(* IEC 61131-3 sources: SmartHomeNew/ (part 7) *)

(* ---- FB_Heating_Source_Stability_Observer.st ---- *)
// ==============================================================================
// Heating source stability observer
//
// Predictive observability-only layer.
//
// DOES NOT own runtime authority.
// DOES NOT own outputs.
// DOES NOT close valves.
// DOES NOT modify heating demand.
// DOES NOT override runtime decisions.
//
// Observes:
// - source switching frequency
// - fallback oscillation
// - degradation persistence
// - recovery trends
// - confidence volatility
//
// Publishes predictive instability semantics only.
//
// Reads only canonical runtime projection contracts.
// Does not depend on explainability publication topology.
// ==============================================================================
FUNCTION_BLOCK FB_Heating_Source_Stability_Observer
VAR_INPUT
    VI_Enable : BOOL;
    VI_System_Time_MS : UDINT;
END_VAR

VAR
    L_i : INT;

    L_Last_Confidence : ARRAY[1..GVL_CONSTANTS.C_MAX_HEATING_CIRCUITS] OF REAL;

    L_Confidence_Delta : REAL;
    L_Confidence_Volatility : REAL;
    L_Source_Trust_Trend : REAL;
    L_Instability_Score : REAL;
END_VAR

IF NOT VI_Enable THEN
    RETURN;
END_IF;

FOR L_i := 1 TO GVL_CONSTANTS.C_MAX_HEATING_CIRCUITS DO

    // ======================================================
    // VISIBILITY
    // ======================================================
    GVL_Heating_Source_Stability.G_State[L_i].Visible :=
        GVL_Heating_Runtime_Projection.G_Circuit_Projection[L_i].Visible;

    // ======================================================
    // EDGE COUNTING
    // ======================================================
    IF GVL_Heating_Runtime_Projection.G_Circuit_Projection[L_i].Source_Switched_Event THEN
        IF GVL_Heating_Source_Stability.G_State[L_i].Source_Switch_Count < 65535 THEN
            GVL_Heating_Source_Stability.G_State[L_i].Source_Switch_Count :=
                GVL_Heating_Source_Stability.G_State[L_i].Source_Switch_Count + 1;
        END_IF;

        GVL_Heating_Source_Stability.G_State[L_i].Last_Observation_MS :=
            VI_System_Time_MS;
    END_IF;

    IF GVL_Heating_Runtime_Projection.G_Circuit_Projection[L_i].Fallback_Activated_Event THEN
        IF GVL_Heating_Source_Stability.G_State[L_i].Fallback_Activation_Count < 65535 THEN
            GVL_Heating_Source_Stability.G_State[L_i].Fallback_Activation_Count :=
                GVL_Heating_Source_Stability.G_State[L_i].Fallback_Activation_Count + 1;
        END_IF;

        GVL_Heating_Source_Stability.G_State[L_i].Last_Observation_MS :=
            VI_System_Time_MS;
    END_IF;

    IF GVL_Heating_Runtime_Projection.G_Circuit_Projection[L_i].Fallback_Recovered_Event THEN
        IF GVL_Heating_Source_Stability.G_State[L_i].Fallback_Recovery_Count < 65535 THEN
            GVL_Heating_Source_Stability.G_State[L_i].Fallback_Recovery_Count :=
                GVL_Heating_Source_Stability.G_State[L_i].Fallback_Recovery_Count + 1;
        END_IF;

        GVL_Heating_Source_Stability.G_State[L_i].Last_Observation_MS :=
            VI_System_Time_MS;
    END_IF;

    IF GVL_Heating_Runtime_Projection.G_Circuit_Projection[L_i].Source_Loss_Event THEN
        IF GVL_Heating_Source_Stability.G_State[L_i].Source_Loss_Count < 65535 THEN
            GVL_Heating_Source_Stability.G_State[L_i].Source_Loss_Count :=
                GVL_Heating_Source_Stability.G_State[L_i].Source_Loss_Count + 1;
        END_IF;

        GVL_Heating_Source_Stability.G_State[L_i].Last_Observation_MS :=
            VI_System_Time_MS;
    END_IF;

    // ======================================================
    // CONFIDENCE VOLATILITY
    // ======================================================
    L_Confidence_Delta := ABS(
        GVL_Heating_Runtime_Projection.G_Circuit_Projection[L_i].Selected_Source_Confidence -
        L_Last_Confidence[L_i]
    );

    L_Confidence_Volatility :=
        GVL_Heating_Source_Stability.G_State[L_i].Confidence_Volatility * REAL#0.90 +
        L_Confidence_Delta * REAL#0.10;

    IF L_Confidence_Volatility < REAL#0.0 THEN
        L_Confidence_Volatility := REAL#0.0;
    ELSIF L_Confidence_Volatility > REAL#1.0 THEN
        L_Confidence_Volatility := REAL#1.0;
    END_IF;

    GVL_Heating_Source_Stability.G_State[L_i].Confidence_Volatility :=
        L_Confidence_Volatility;

    // ======================================================
    // SOURCE TRUST TREND
    // ======================================================
    L_Source_Trust_Trend :=
        GVL_Heating_Source_Stability.G_State[L_i].Source_Trust_Trend * REAL#0.95 +
        GVL_Heating_Runtime_Projection.G_Circuit_Projection[L_i].Selected_Source_Confidence * REAL#0.05;

    IF GVL_Heating_Runtime_Projection.G_Circuit_Projection[L_i].Source_Degraded THEN
        L_Source_Trust_Trend := L_Source_Trust_Trend * REAL#0.98;
    END_IF;

    IF L_Source_Trust_Trend < REAL#0.0 THEN
        L_Source_Trust_Trend := REAL#0.0;
    ELSIF L_Source_Trust_Trend > REAL#1.0 THEN
        L_Source_Trust_Trend := REAL#1.0;
    END_IF;

    GVL_Heating_Source_Stability.G_State[L_i].Source_Trust_Trend :=
        L_Source_Trust_Trend;

    // ======================================================
    // TREND OBSERVATION
    // ======================================================
    GVL_Heating_Source_Stability.G_State[L_i].Degraded_Trend_Visible :=
        GVL_Heating_Runtime_Projection.G_Circuit_Projection[L_i].Source_Degraded OR
        (GVL_Heating_Source_Stability.G_State[L_i].Fallback_Activation_Count >
         GVL_Heating_Source_Stability.G_State[L_i].Fallback_Recovery_Count);

    GVL_Heating_Source_Stability.G_State[L_i].Recovery_Trend_Visible :=
        (GVL_Heating_Source_Stability.G_State[L_i].Fallback_Recovery_Count > 0) AND
        (GVL_Heating_Source_Stability.G_State[L_i].Fallback_Recovery_Count >=
         GVL_Heating_Source_Stability.G_State[L_i].Fallback_Activation_Count);

    GVL_Heating_Source_Stability.G_State[L_i].Oscillation_Detected :=
        (GVL_Heating_Source_Stability.G_State[L_i].Source_Switch_Count >= 3) OR
        ((GVL_Heating_Source_Stability.G_State[L_i].Fallback_Activation_Count >= 2) AND
         (GVL_Heating_Source_Stability.G_State[L_i].Fallback_Recovery_Count >= 2));

    // ======================================================
    // INSTABILITY SCORE
    // ======================================================
    L_Instability_Score := REAL#0.0;

    IF GVL_Heating_Source_Stability.G_State[L_i].Oscillation_Detected THEN
        L_Instability_Score := L_Instability_Score + REAL#40.0;
    END_IF;

    IF GVL_Heating_Source_Stability.G_State[L_i].Degraded_Trend_Visible THEN
        L_Instability_Score := L_Instability_Score + REAL#30.0;
    END_IF;

    IF GVL_Heating_Source_Stability.G_State[L_i].Source_Loss_Count > 0 THEN
        L_Instability_Score := L_Instability_Score + REAL#30.0;
    END_IF;

    L_Instability_Score :=
        L_Instability_Score +
        (GVL_Heating_Source_Stability.G_State[L_i].Confidence_Volatility * REAL#20.0);

    IF L_Instability_Score > REAL#100.0 THEN
        L_Instability_Score := REAL#100.0;
    END_IF;

    GVL_Heating_Source_Stability.G_State[L_i].Instability_Score :=
        L_Instability_Score;

    GVL_Heating_Source_Stability.G_State[L_i].Instability_Attention :=
        L_Instability_Score >= REAL#60.0;

    // ======================================================
    // EXPLAINABILITY PUBLICATION
    // ======================================================
    IF GVL_Heating_Source_Stability.G_State[L_i].Source_Loss_Count > 0 THEN
        GVL_Heating_Source_Stability.G_State[L_i].Status_Code := 904;
        GVL_Heating_Source_Stability.G_State[L_i].Status_Text :=
            'Predictive source instability: source loss observed';

    ELSIF GVL_Heating_Source_Stability.G_State[L_i].Oscillation_Detected THEN
        GVL_Heating_Source_Stability.G_State[L_i].Status_Code := 903;
        GVL_Heating_Source_Stability.G_State[L_i].Status_Text :=
            'Predictive source instability: oscillation detected';

    ELSIF GVL_Heating_Source_Stability.G_State[L_i].Degraded_Trend_Visible THEN
        GVL_Heating_Source_Stability.G_State[L_i].Status_Code := 902;
        GVL_Heating_Source_Stability.G_State[L_i].Status_Text :=
            'Predictive source degradation trend observed';

    ELSE
        GVL_Heating_Source_Stability.G_State[L_i].Status_Code := 901;
        GVL_Heating_Source_Stability.G_State[L_i].Status_Text :=
            'Source stability nominal';
    END_IF;

    L_Last_Confidence[L_i] :=
        GVL_Heating_Runtime_Projection.G_Circuit_Projection[L_i].Selected_Source_Confidence;
END_FOR;

END_FUNCTION_BLOCK
// >>> BULK_SYNC_ANCHOR: FB_Heating_Source_Stability_Observer <<<

(* ---- FB_Heating_System_Manager.st ---- *)
FUNCTION_BLOCK FB_Heating_System_Manager
VAR_INPUT
    VI_System_Mode : E_System_Operating_Mode;
    VI_System_Time_MS : UDINT;
    VI_IsActivePLC : BOOL;
    VI_Outdoor_Temp : REAL;
    VI_Config : ST_Heating_Config;
    VI_Tariff : ST_Tariff_Config;
    VI_Current_Hour : UINT;
    VI_DHW_Heating_Demand : BOOL;
    VI_DHW_Target_Temp : REAL;
    VI_Emergency_Stop : BOOL;
    VI_Gas_Safety_Stop : BOOL;
    VI_Boiler_Error_Status : ARRAY[1..GVL_CONSTANTS.C_MAX_BOILERS] OF BOOL;
    VI_Boiler_OT_Online : ARRAY[1..GVL_CONSTANTS.C_MAX_BOILERS] OF BOOL;
    VI_Boiler_Modulation : ARRAY[1..GVL_CONSTANTS.C_MAX_BOILERS] OF REAL;
END_VAR
VAR_IN_OUT
    VI_Floor_Temps : ARRAY[1..GVL_CONSTANTS.C_MAX_HEATING_CIRCUITS] OF REAL;
    VI_Room_Temps : ARRAY[1..GVL_CONSTANTS.C_MAX_ZONES] OF REAL;
    VI_Manifold_Pressures : ARRAY[1..GVL_CONSTANTS.C_MAX_MANIFOLDS] OF REAL;
    VI_Manifold_Currents : ARRAY[1..GVL_CONSTANTS.C_MAX_MANIFOLDS] OF REAL;
    VI_Manifold_Temps_Supply : ARRAY[1..GVL_CONSTANTS.C_MAX_MANIFOLDS] OF REAL;
    VI_Manifold_Temps_Return : ARRAY[1..GVL_CONSTANTS.C_MAX_MANIFOLDS] OF REAL;
    VI_Boiler_Flame_Status : ARRAY[1..GVL_CONSTANTS.C_MAX_BOILERS] OF BOOL;
    VI_Zone_Configs : ARRAY[1..GVL_CONSTANTS.C_MAX_HEATING_CIRCUITS] OF ST_FloorHeating_Circuit_Config;
    VI_Rule_Actions : ARRAY[1..GVL_CONSTANTS.C_MAX_RULES] OF ST_Rule_Action;
    VI_IO_Modules_Online : ARRAY[1..GVL_CONSTANTS.C_MAX_MODULES] OF BOOL;
    VI_Manifold_End_Switches : ARRAY[1..GVL_CONSTANTS.C_MAX_MANIFOLDS] OF BOOL;
    VI_Valve_Test_Config : ARRAY[1..GVL_CONSTANTS.C_MAX_MANIFOLDS] OF ST_Valve_Test_Config;
END_VAR
VAR_OUTPUT
    VO_Manifold_Valves : ARRAY[1..GVL_CONSTANTS.C_MAX_MANIFOLDS] OF REAL;
    VO_Manifold_Pumps : ARRAY[1..GVL_CONSTANTS.C_MAX_MANIFOLDS] OF BOOL;
    VO_Zone_Valves : ARRAY[1..GVL_CONSTANTS.C_MAX_HEATING_CIRCUITS] OF BOOL;
    VO_Boiler_OT_Enable : ARRAY[1..GVL_CONSTANTS.C_MAX_BOILERS] OF BOOL;
    VO_Boiler_OT_Setpoint : ARRAY[1..GVL_CONSTANTS.C_MAX_BOILERS] OF REAL;
    VO_Backup_Circulation_Pump : BOOL;
    VO_Electric_Heater_Enable : BOOL;
    VO_Freeze_Risk_Status : BOOL;
    VO_Status : ARRAY[1..GVL_CONSTANTS.C_MAX_MANIFOLDS] OF ST_Manifold_Status;
    VO_Boiler_Status : ARRAY[1..GVL_CONSTANTS.C_MAX_BOILERS] OF ST_Boiler_Status;
END_VAR
VAR
    L_i : INT;
    L_Target_Supply_Temp : REAL;
    L_Manifold_Demand_Map : ARRAY[1..GVL_CONSTANTS.C_MAX_MANIFOLDS] OF BOOL;
    L_Manifold_Demand_Filtered : ARRAY[1..GVL_CONSTANTS.C_MAX_MANIFOLDS] OF BOOL;
    L_Manifold_Available : ARRAY[1..GVL_CONSTANTS.C_MAX_MANIFOLDS] OF BOOL;
    L_Manifold_In_Service : ARRAY[1..GVL_CONSTANTS.C_MAX_MANIFOLDS] OF BOOL;
    L_Manifold_Subsystem_Degraded : ARRAY[1..GVL_CONSTANTS.C_MAX_MANIFOLDS] OF BOOL;
    L_Manifold_Base_Priority : ARRAY[1..GVL_CONSTANTS.C_MAX_MANIFOLDS] OF INT;
    L_Manifold_Thermal_Weight : ARRAY[1..GVL_CONSTANTS.C_MAX_MANIFOLDS] OF REAL;
    L_Allocation_Degraded : BOOL;
    fbValveTestManager : FB_Valve_Test_Manager;
    L_IO_Failsafe_Active : BOOL;
    L_Freeze_Active : BOOL;
    L_Freeze_Target_Supply : REAL;
    L_Policy_Degraded : BOOL;
    L_Sensor_Error : BOOL;
    L_Subsys_Degraded : BOOL;
    L_Pressure_OK : BOOL;
    L_Prev_Pressure : ARRAY[1..GVL_CONSTANTS.C_MAX_MANIFOLDS] OF REAL;
    L_Prev_Current : ARRAY[1..GVL_CONSTANTS.C_MAX_MANIFOLDS] OF REAL;
    L_Error_Instant : REAL;
    L_Confidence : REAL;
    fbAdaptiveTarget : FB_Heating_Adaptive_Target;
    fbSafetyGate : FB_Heating_Safety_Gate;
    fbSafeState : FB_Heating_Safe_State;
    fbDemandMap : FB_Heating_Demand_Map;
    fbAllocationFilter : FB_Heating_Allocation_Filter;
    fbCircuitControl : FB_Heating_Circuit_Control;
    fbManifoldControl : FB_Heating_Manifold_Control;
    fbBoilerControl : FB_Heating_Boiler_Control;
END_VAR

L_Policy_Degraded := (VI_System_Mode = E_System_Operating_Mode.MODE_DEGRADED);

GVL_STATE.G_Heating_IO_Fault := FALSE;
GVL_STATE.G_Heating_Sensor_Fault := FALSE;
GVL_STATE.G_Heating_Subsystem_Degraded := FALSE;
L_Sensor_Error := FALSE;
L_Subsys_Degraded := FALSE;
L_Allocation_Degraded := FALSE;

L_IO_Failsafe_Active := FALSE;
FOR L_i := 1 TO GVL_CONSTANTS.C_MAX_MODULES DO
    IF NOT VI_IO_Modules_Online[L_i] THEN
        L_IO_Failsafe_Active := TRUE;
        GVL_STATE.G_Heating_IO_Fault := TRUE;
        GVL_STATE.G_Heating_Subsystem_Degraded := TRUE;
        EXIT;
    END_IF;
END_FOR;

fbSafetyGate(
    VI_System_Mode := VI_System_Mode,
    VI_Emergency_Stop := VI_Emergency_Stop,
    VI_Gas_Safety_Stop := VI_Gas_Safety_Stop,
    VI_IO_Failsafe_Active := L_IO_Failsafe_Active,
    VI_Outdoor_Temp := VI_Outdoor_Temp,
    VI_Freeze_Threshold := VI_Config.Freeze_Threshold,
    VI_Floor_Temps := VI_Floor_Temps,
    VO_Freeze_Mode_Active => L_Freeze_Active,
    VO_Freeze_Target_Supply => L_Freeze_Target_Supply
);

fbSafeState(
    VI_Block_Normal_Heating := fbSafetyGate.VO_Block_Normal_Heating,
    VI_IO_Failsafe_Active := fbSafetyGate.VO_IO_Failsafe_Active,
    VI_Gas_Safety_Active := fbSafetyGate.VO_Gas_Safety_Active,
    VI_Freeze_Active := L_Freeze_Active,
    VI_Freeze_Target_Supply := L_Freeze_Target_Supply,
    VI_Manifold_Temps_Supply := VI_Manifold_Temps_Supply,
    VI_Boiler_Error_Status := VI_Boiler_Error_Status,
    VI_Boiler_OT_Online := VI_Boiler_OT_Online
);

IF fbSafeState.VO_Applied THEN
    FOR L_i := 1 TO GVL_CONSTANTS.C_MAX_HEATING_CIRCUITS DO
        VO_Zone_Valves[L_i] := fbSafeState.VO_Zone_Valves[L_i];
    END_FOR;

    FOR L_i := 1 TO GVL_CONSTANTS.C_MAX_MANIFOLDS DO
        VO_Manifold_Pumps[L_i] := fbSafeState.VO_Manifold_Pumps[L_i];
        VO_Manifold_Valves[L_i] := fbSafeState.VO_Manifold_Valves[L_i];
    END_FOR;

    FOR L_i := 1 TO GVL_CONSTANTS.C_MAX_BOILERS DO
        VO_Boiler_OT_Enable[L_i] := fbSafeState.VO_Boiler_OT_Enable[L_i];
        VO_Boiler_OT_Setpoint[L_i] := fbSafeState.VO_Boiler_OT_Setpoint[L_i];
        VO_Boiler_Status[L_i] := fbSafeState.VO_Boiler_Status[L_i];
    END_FOR;

    VO_Backup_Circulation_Pump := fbSafeState.VO_Backup_Circulation_Pump;
    VO_Electric_Heater_Enable := fbSafeState.VO_Electric_Heater_Enable;
    VO_Freeze_Risk_Status := fbSafeState.VO_Freeze_Risk_Status;
    RETURN;
END_IF;

VO_Backup_Circulation_Pump := FALSE;
VO_Electric_Heater_Enable := FALSE;
VO_Freeze_Risk_Status := FALSE;

IF L_Freeze_Active THEN
    L_Target_Supply_Temp := L_Freeze_Target_Supply;
ELSE
    L_Target_Supply_Temp := VI_Config.Target_Floor_Temp;
END_IF;

fbAdaptiveTarget(
    VI_Base_Target_Supply_Temp := L_Target_Supply_Temp,
    VI_Global_Target_Temperature := GVL_STATE.G_Target_Temperature,
    VI_Zone_Configs := VI_Zone_Configs,
    VI_Floor_Temps := VI_Floor_Temps,
    VI_Room_Temps := VI_Room_Temps,
    VO_Target_Supply_Temp => L_Target_Supply_Temp
);

fbCircuitControl(
    VI_System_Time_MS := VI_System_Time_MS,
    VI_Current_Hour := VI_Current_Hour,
    VI_IsActivePLC := VI_IsActivePLC,
    VI_Config := VI_Config,
    VI_Tariff := VI_Tariff,
    VI_Scenario_Adjust := REAL#0.0,
    VI_Zone_Configs := VI_Zone_Configs,
    VI_Floor_Temps := VI_Floor_Temps,
    VI_Room_Temps := VI_Room_Temps,
    VI_Rule_Actions := VI_Rule_Actions,
    VO_Zone_Valves => VO_Zone_Valves,
    VO_Heating_Sensor_Fault => L_Sensor_Error
);

GVL_STATE.G_Heating_Sensor_Fault := L_Sensor_Error;

fbDemandMap(
    VI_Zone_Valves := VO_Zone_Valves,
    VI_Zone_Configs := VI_Zone_Configs,
    VO_Manifold_Demand_Map => L_Manifold_Demand_Map
);

FOR L_i := 1 TO GVL_CONSTANTS.C_MAX_MANIFOLDS DO
    L_Manifold_Available[L_i] := VI_Manifold_Pressures[L_i] >= GVL_CONSTANTS.C_MIN_HEATING_MANIFOLD_PRESSURE;
    L_Manifold_In_Service[L_i] := GVL_CONFIG.G_Manifold_Pump_In_Service[L_i];
    L_Manifold_Subsystem_Degraded[L_i] :=
        GVL_STATE.G_Predictive_Pump_Pressure_Drop[L_i]
        OR GVL_STATE.G_Predictive_Pump_Current_Rise[L_i];
    L_Manifold_Base_Priority[L_i] := 0;
    L_Manifold_Thermal_Weight[L_i] := REAL#1.0;
END_FOR;

fbAllocationFilter(
    VI_Enable := TRUE,
    VI_Enable_Policy_Allocation := FALSE,
    VI_Freeze_Mode_Active := L_Freeze_Active,
    VI_DHW_Heating_Demand := VI_DHW_Heating_Demand,
    VI_Manifold_Demand_Map := L_Manifold_Demand_Map,
    VI_Manifold_Available := L_Manifold_Available,
    VI_Manifold_In_Service := L_Manifold_In_Service,
    VI_Manifold_Subsystem_Degraded := L_Manifold_Subsystem_Degraded,
    VI_Manifold_Base_Priority := L_Manifold_Base_Priority,
    VI_Manifold_Thermal_Weight := L_Manifold_Thermal_Weight,
    VI_Max_Thermal_Budget := REAL#0.0,
    VO_Manifold_Demand_Filtered => L_Manifold_Demand_Filtered,
    VO_Allocation_Degraded => L_Allocation_Degraded
);

IF L_Allocation_Degraded THEN
    GVL_STATE.G_Heating_Subsystem_Degraded := TRUE;
END_IF;

fbManifoldControl(
    VI_System_Time_MS := VI_System_Time_MS,
    VI_IsActivePLC := VI_IsActivePLC,
    VI_DHW_Heating_Demand := VI_DHW_Heating_Demand,
    VI_Freeze_Mode_Active := L_Freeze_Active,
    VI_Target_Supply_Temp := L_Target_Supply_Temp,
    VI_Any_Zone_Active := L_Manifold_Demand_Filtered,
    VI_Manifold_Pressures := VI_Manifold_Pressures,
    VI_Manifold_Currents := VI_Manifold_Currents,
    VI_Manifold_Temps_Supply := VI_Manifold_Temps_Supply,
    VI_Manifold_Temps_Return := VI_Manifold_Temps_Return,
    VO_Manifold_Pumps => VO_Manifold_Pumps,
    VO_Manifold_Valves => VO_Manifold_Valves,
    VO_Status => VO_Status
);

FOR L_i := 1 TO GVL_CONSTANTS.C_MAX_MANIFOLDS DO
    L_Pressure_OK := VI_Manifold_Pressures[L_i] >= GVL_CONSTANTS.C_MIN_HEATING_MANIFOLD_PRESSURE;

    IF VO_Manifold_Pumps[L_i] AND NOT L_Pressure_OK THEN
        VO_Manifold_Pumps[L_i] := FALSE;
        GVL_STATE.G_Heating_Subsystem_Degraded := TRUE;
    END_IF;

    IF (L_Prev_Pressure[L_i] > REAL#0.0) AND ((L_Prev_Pressure[L_i] - VI_Manifold_Pressures[L_i]) > REAL#0.2) THEN
        GVL_STATE.G_Predictive_Pump_Pressure_Drop[L_i] := TRUE;
    ELSE
        GVL_STATE.G_Predictive_Pump_Pressure_Drop[L_i] := FALSE;
    END_IF;

    IF (L_Prev_Current[L_i] > REAL#0.0) AND (VI_Manifold_Currents[L_i] > (L_Prev_Current[L_i] * REAL#1.2)) THEN
        GVL_STATE.G_Predictive_Pump_Current_Rise[L_i] := TRUE;
    ELSE
        GVL_STATE.G_Predictive_Pump_Current_Rise[L_i] := FALSE;
    END_IF;

    IF GVL_STATE.G_Predictive_Pump_Pressure_Drop[L_i] OR GVL_STATE.G_Predictive_Pump_Current_Rise[L_i] THEN
        GVL_STATE.G_Heating_Subsystem_Degraded := TRUE;
    END_IF;

    L_Prev_Pressure[L_i] := VI_Manifold_Pressures[L_i];
    L_Prev_Current[L_i] := VI_Manifold_Currents[L_i];
END_FOR;

L_Error_Instant := REAL#0.0;

IF GVL_STATE.G_Heating_Sensor_Fault THEN
    L_Error_Instant := L_Error_Instant + REAL#0.2;
END_IF;

IF GVL_STATE.G_Heating_IO_Fault THEN
    L_Error_Instant := L_Error_Instant + REAL#0.2;
END_IF;

FOR L_i := 1 TO GVL_CONSTANTS.C_MAX_MANIFOLDS DO
    IF VI_Manifold_Pressures[L_i] < GVL_CONSTANTS.C_MIN_HEATING_MANIFOLD_PRESSURE THEN
        L_Error_Instant := L_Error_Instant + REAL#0.1;
        EXIT;
    END_IF;
END_FOR;

FOR L_i := 1 TO GVL_CONSTANTS.C_MAX_MANIFOLDS DO
    IF GVL_STATE.G_Predictive_Pump_Pressure_Drop[L_i] OR GVL_STATE.G_Predictive_Pump_Current_Rise[L_i] THEN
        L_Error_Instant := L_Error_Instant + REAL#0.2;
        EXIT;
    END_IF;
END_FOR;

GVL_STATE.G_Heating_Error_Score := (GVL_STATE.G_Heating_Error_Score * REAL#0.98) + L_Error_Instant;
L_Confidence := REAL#1.0 - GVL_STATE.G_Heating_Error_Score;

IF L_Confidence < REAL#0.0 THEN
    L_Confidence := REAL#0.0;
ELSIF L_Confidence > REAL#1.0 THEN
    L_Confidence := REAL#1.0;
END_IF;

GVL_STATE.G_Heating_Confidence := L_Confidence;

GVL_STATE.G_Heating_Confidence_Reason_Code := 0;
GVL_STATE.G_Heating_Confidence_Reason_Text := 'OK';

IF GVL_STATE.G_Heating_IO_Fault THEN
    GVL_STATE.G_Heating_Confidence_Reason_Code := 2;
    GVL_STATE.G_Heating_Confidence_Reason_Text := 'IO fault detected';
ELSIF GVL_STATE.G_Heating_Sensor_Fault THEN
    GVL_STATE.G_Heating_Confidence_Reason_Code := 1;
    GVL_STATE.G_Heating_Confidence_Reason_Text := 'Sensor fault detected';
ELSE
    FOR L_i := 1 TO GVL_CONSTANTS.C_MAX_MANIFOLDS DO
        IF VI_Manifold_Pressures[L_i] < GVL_CONSTANTS.C_MIN_HEATING_MANIFOLD_PRESSURE THEN
            GVL_STATE.G_Heating_Confidence_Reason_Code := 3;
            GVL_STATE.G_Heating_Confidence_Reason_Text := 'Low manifold pressure';
            EXIT;
        END_IF;
    END_FOR;

    FOR L_i := 1 TO GVL_CONSTANTS.C_MAX_MANIFOLDS DO
        IF GVL_STATE.G_Predictive_Pump_Pressure_Drop[L_i] OR GVL_STATE.G_Predictive_Pump_Current_Rise[L_i] THEN
            GVL_STATE.G_Heating_Confidence_Reason_Code := 4;
            GVL_STATE.G_Heating_Confidence_Reason_Text := 'Predictive pump degradation';
            EXIT;
        END_IF;
    END_FOR;
END_IF;

IF GVL_STATE.G_Heating_Confidence < REAL#0.5 THEN
    L_Target_Supply_Temp := L_Target_Supply_Temp - REAL#3.0;
END_IF;

CASE GVL_STATE.G_Heating_Confidence_Reason_Code OF
    1:
        L_Target_Supply_Temp := LIMIT(GVL_CONSTANTS.C_BOILER_SETPOINT_MIN, REAL#40.0, GVL_CONSTANTS.C_BOILER_SETPOINT_MAX);
    2:
        VO_Backup_Circulation_Pump := TRUE;
    3:
        FOR L_i := 1 TO GVL_CONSTANTS.C_MAX_MANIFOLDS DO
            VO_Manifold_Pumps[L_i] := FALSE;
        END_FOR;
    4:
        L_Target_Supply_Temp := LIMIT(GVL_CONSTANTS.C_BOILER_SETPOINT_MIN, L_Target_Supply_Temp - REAL#5.0, GVL_CONSTANTS.C_BOILER_SETPOINT_MAX);
ELSE
    // no auto-recovery action
END_CASE;

fbValveTestManager(
    VI_System_Time_MS := VI_System_Time_MS,
    VI_IsActivePLC := VI_IsActivePLC,
    VI_Valve_Currents := VI_Manifold_Currents,
    VI_Valve_End_Switches := VI_Manifold_End_Switches,
    VI_Config := VI_Valve_Test_Config
);

IF fbValveTestManager.VO_Test_Active THEN
    L_i := fbValveTestManager.VO_Current_Valve;
    IF L_i >= 1 AND L_i <= GVL_CONSTANTS.C_MAX_MANIFOLDS THEN
        IF fbValveTestManager.VO_Valve_Cmd[L_i] THEN
            VO_Manifold_Valves[L_i] := REAL#100.0;
        ELSE
            VO_Manifold_Valves[L_i] := REAL#0.0;
        END_IF;
        VO_Manifold_Pumps[L_i] := FALSE;
    END_IF;
END_IF;

fbBoilerControl(
    VI_System_Time_MS := VI_System_Time_MS,
    VI_IsActivePLC := VI_IsActivePLC,
    VI_DHW_Heating_Demand := VI_DHW_Heating_Demand,
    VI_DHW_Target_Temp := VI_DHW_Target_Temp,
    VI_Target_Supply_Temp := L_Target_Supply_Temp,
    VI_Freeze_Mode_Active := L_Freeze_Active,
    VI_Policy_Degraded := L_Policy_Degraded,
    VI_Manifold_Pumps := VO_Manifold_Pumps,
    VI_Manifold_Valves := VO_Manifold_Valves,
    VI_Boiler_Flame_Status := VI_Boiler_Flame_Status,
    VI_Boiler_Error_Status := VI_Boiler_Error_Status,
    VI_Boiler_OT_Online := VI_Boiler_OT_Online,
    VI_Boiler_Modulation := VI_Boiler_Modulation,
    VO_Boiler_OT_Enable => VO_Boiler_OT_Enable,
    VO_Boiler_OT_Setpoint => VO_Boiler_OT_Setpoint,
    VO_Boiler_Status => VO_Boiler_Status,
    VO_Any_Subsystem_Degraded => L_Subsys_Degraded
);

GVL_STATE.G_Heating_Subsystem_Degraded := GVL_STATE.G_Heating_Subsystem_Degraded OR L_Subsys_Degraded;

END_FUNCTION_BLOCK
// >>> BULK_SYNC_ANCHOR: FB_Heating_System_Manager <<<

(* ---- FB_Heating_Thermal_Allocation.st ---- *)
FUNCTION_BLOCK FB_Heating_Thermal_Allocation
VAR_INPUT
    VI_Zone_Configs : ARRAY[1..GVL_CONSTANTS.C_MAX_HEATING_CIRCUITS] OF ST_FloorHeating_Circuit_Config;
    VI_Circuit_To_Zone : ARRAY[1..GVL_CONSTANTS.C_MAX_HEATING_CIRCUITS] OF INT;
    VI_Manifold_Base_Priority : ARRAY[1..GVL_CONSTANTS.C_MAX_MANIFOLDS] OF INT;
    VI_Zone_Priority_Bias : ARRAY[1..GVL_CONSTANTS.C_MAX_ZONES] OF REAL;
    VI_Guest_Preheat_Enabled : BOOL;
    VI_Zone_Guest_Preheat_Request : ARRAY[1..GVL_CONSTANTS.C_MAX_ZONES] OF BOOL;
    VI_Guest_Preheat_Priority_Boost : INT;
    VI_Zone_Target_Adjustment : ARRAY[1..GVL_CONSTANTS.C_MAX_ZONES] OF REAL;
    VI_Zone_Self_Level : ARRAY[1..GVL_CONSTANTS.C_MAX_ZONES] OF INT;
    VI_Policy_Priority_Multiplier : REAL;
    VI_Manifold_Pump_In_Service : ARRAY[1..GVL_CONSTANTS.C_MAX_MANIFOLDS] OF BOOL;
    VI_Manifold_Pressure_Fault : ARRAY[1..GVL_CONSTANTS.C_MAX_MANIFOLDS] OF BOOL;
    VI_Manifold_Current_Fault : ARRAY[1..GVL_CONSTANTS.C_MAX_MANIFOLDS] OF BOOL;
    VI_Manifold_Thermal_Weight : ARRAY[1..GVL_CONSTANTS.C_MAX_MANIFOLDS] OF REAL;
    VI_Max_Thermal_Budget : REAL;
END_VAR
VAR_OUTPUT
    VO_Manifold_Adjusted_Priority : ARRAY[1..GVL_CONSTANTS.C_MAX_MANIFOLDS] OF INT;
    VO_Manifold_Allowed : ARRAY[1..GVL_CONSTANTS.C_MAX_MANIFOLDS] OF BOOL;
    VO_Manifold_Enabled : ARRAY[1..GVL_CONSTANTS.C_MAX_MANIFOLDS] OF BOOL;
    VO_Heating_Degraded : BOOL;
END_VAR
VAR
    fbDecision : FB_Heating_Decision_Context;
    L_i : INT;
    L_j : INT;
    L_Zone_ID : INT;
END_VAR

// Extracted candidate from PRG_Heating S1.5
// Not connected yet.

// Base copy
FOR L_i := 1 TO GVL_CONSTANTS.C_MAX_MANIFOLDS DO
    VO_Manifold_Adjusted_Priority[L_i] := VI_Manifold_Base_Priority[L_i];
END_FOR;

// Adjustment loop
FOR L_i := 1 TO GVL_CONSTANTS.C_MAX_HEATING_CIRCUITS DO

    L_j := TO_INT(VI_Zone_Configs[L_i].manifold_id);
    L_Zone_ID := VI_Circuit_To_Zone[L_i];

    IF (L_j >= 1) AND (L_j <= GVL_CONSTANTS.C_MAX_MANIFOLDS) AND
       (L_Zone_ID >= 1) AND (L_Zone_ID <= GVL_CONSTANTS.C_MAX_ZONES) THEN

        VO_Manifold_Adjusted_Priority[L_j] := VO_Manifold_Adjusted_Priority[L_j]
            + TO_INT(VI_Zone_Priority_Bias[L_Zone_ID]);

        IF VI_Guest_Preheat_Enabled AND VI_Zone_Guest_Preheat_Request[L_Zone_ID] THEN
            VO_Manifold_Adjusted_Priority[L_j] := VO_Manifold_Adjusted_Priority[L_j]
                + VI_Guest_Preheat_Priority_Boost;
        END_IF;

        IF VI_Zone_Target_Adjustment[L_Zone_ID] > 0.1 THEN
            VO_Manifold_Adjusted_Priority[L_j] := VO_Manifold_Adjusted_Priority[L_j] + 1;
        ELSIF VI_Zone_Target_Adjustment[L_Zone_ID] < -0.1 THEN
            VO_Manifold_Adjusted_Priority[L_j] := VO_Manifold_Adjusted_Priority[L_j] - 1;
        END_IF;

        VO_Manifold_Adjusted_Priority[L_j] := VO_Manifold_Adjusted_Priority[L_j]
            + VI_Zone_Self_Level[L_Zone_ID];

        VO_Manifold_Adjusted_Priority[L_j] := TO_INT(
            TO_REAL(VO_Manifold_Adjusted_Priority[L_j])
            * VI_Policy_Priority_Multiplier
        );

        IF VO_Manifold_Adjusted_Priority[L_j] < 1 THEN
            VO_Manifold_Adjusted_Priority[L_j] := 1;
        END_IF;

    END_IF;

END_FOR;

// Decision context call
fbDecision(
    VI_Manifold_Pump_In_Service := VI_Manifold_Pump_In_Service,
    VI_Manifold_Pressure_Fault := VI_Manifold_Pressure_Fault,
    VI_Manifold_Current_Fault := VI_Manifold_Current_Fault,
    VI_Manifold_Thermal_Weight := VI_Manifold_Thermal_Weight,
    VI_Manifold_Priority := VO_Manifold_Adjusted_Priority,
    VI_Max_Thermal_Budget := VI_Max_Thermal_Budget
);

VO_Manifold_Allowed := fbDecision.VO_Manifold_Allowed;
VO_Manifold_Enabled := fbDecision.VO_Manifold_Enabled;
VO_Heating_Degraded := fbDecision.VO_Heating_Degraded;

END_FUNCTION_BLOCK
// >>> BULK_SYNC_ANCHOR: FB_Heating_Thermal_Allocation <<<

(* ---- FB_Heating_Thermal_Model.st ---- *)
FUNCTION_BLOCK FB_Heating_Thermal_Model
VAR
    L_i : INT;
    L_DeltaT : REAL;
    L_Loss : REAL;
    L_Gain : REAL;
    L_Outdoor : REAL;
END_VAR

L_Outdoor := GVL_STATE.G_Outdoor_Temp;

FOR L_i := 1 TO GVL_CONSTANTS.C_MAX_ZONES DO

    L_DeltaT := GVL_STATE.G_Room_Temps[L_i] - L_Outdoor;

    L_Loss := L_DeltaT * 0.01 * GVL_HEATING_POLICY.G_Zone_Thermal_Inertia[L_i];

    L_Gain := (GVL_STATE.G_Floor_Temps[L_i] - GVL_STATE.G_Room_Temps[L_i]) * 0.05;

    GVL_HEATING_POLICY.G_Zone_Heat_Loss_Rate[L_i] := L_Loss;
    GVL_HEATING_POLICY.G_Zone_Heat_Gain_Rate[L_i] := L_Gain;

    GVL_HEATING_POLICY.G_Zone_Thermal_Response[L_i] := L_Gain - L_Loss;

    GVL_HEATING_POLICY.G_Zone_Thermal_Demand[L_i] :=
        GVL_STATE.G_Target_Temperature - GVL_STATE.G_Room_Temps[L_i];

    IF ABS(GVL_HEATING_POLICY.G_Zone_Thermal_Response[L_i]) > 0.01 THEN
        GVL_HEATING_POLICY.G_Zone_Time_To_Heat_MS[L_i] :=
            REAL_TO_UDINT(ABS(GVL_HEATING_POLICY.G_Zone_Thermal_Demand[L_i] /
                  GVL_HEATING_POLICY.G_Zone_Thermal_Response[L_i]) * 60000.0);
    ELSE
        GVL_HEATING_POLICY.G_Zone_Time_To_Heat_MS[L_i] := 0;
    END_IF;

    GVL_HEATING_POLICY.G_Zone_Predicted_Temp_30m[L_i] :=
        GVL_STATE.G_Room_Temps[L_i] +
        GVL_HEATING_POLICY.G_Zone_Thermal_Response[L_i] * 30.0;

    GVL_HEATING_POLICY.G_Zone_Thermal_Model_Confidence[L_i] :=
        LIMIT(0.0, 1.0, ABS(GVL_HEATING_POLICY.G_Zone_Thermal_Response[L_i]));

END_FOR;

END_FUNCTION_BLOCK

(* ---- FB_History_Manager.st ---- *)
FUNCTION_BLOCK FB_History_Manager
VAR_INPUT
    VI_System_Time_MS : UDINT;
    VI_Write_Event    : BOOL;
    VI_Event          : ST_History_Record;
END_VAR
VAR_OUTPUT
    VO_Total_Events   : UDINT;
END_VAR

IF VI_Write_Event AND (VI_Event.event_code <> 0) THEN
    GVL_Retain.G_History_Buffer[GVL_Retain.G_History_Write_Idx] := VI_Event;
    GVL_Retain.G_History_Buffer[GVL_Retain.G_History_Write_Idx].timestamp_ms := VI_System_Time_MS;

    GVL_Retain.G_History_Write_Idx := (GVL_Retain.G_History_Write_Idx MOD GVL_CONSTANTS.C_MAX_HISTORY_RECORDS) + 1;
    GVL_Retain.G_History_Total_Events := GVL_Retain.G_History_Total_Events + 1;
END_IF;

VO_Total_Events := GVL_Retain.G_History_Total_Events;
// >>> BULK_SYNC_ANCHOR: FB_History_Manager <<<
END_FUNCTION_BLOCK

(* ---- FB_HMAC_SHA1.st ---- *)
FUNCTION_BLOCK FB_HMAC_SHA1
VAR_INPUT
    KeyLength : INT;
    MessageLength : INT;
END_VAR
VAR_IN_OUT
    Key : ARRAY[0..63] OF BYTE;
    Message : ARRAY[0..7] OF BYTE;
END_VAR
VAR_OUTPUT
    Hash : ARRAY[0..19] OF BYTE;
    Done : BOOL;
END_VAR
VAR
    i : INT;
    K_ipad : ARRAY[0..63] OF BYTE;
    K_opad : ARRAY[0..63] OF BYTE;
    InnerData : ARRAY[0..127] OF BYTE; // 64 (ipad) + 8 (msg)
    OuterData : ARRAY[0..127] OF BYTE; // 64 (opad) + 20 (inner hash)
    InnerHash : ARRAY[0..19] OF BYTE;
    FB_SHA1_Inner : FB_SHA1;
    FB_SHA1_Outer : FB_SHA1;
END_VAR

// 1. Prepare K_ipad and K_opad
FOR i := 0 TO 63 DO
    IF i < KeyLength THEN
        K_ipad[i] := Key[i] XOR 16#36;
        K_opad[i] := Key[i] XOR 16#5C;
    ELSE
        K_ipad[i] := 16#36;
        K_opad[i] := 16#5C;
    END_IF;
END_FOR;

// 2. Inner Hash: SHA1(K_ipad || Message)
FOR i := 0 TO 63 DO
    InnerData[i] := K_ipad[i];
END_FOR;
FOR i := 0 TO MessageLength - 1 DO
    InnerData[64 + i] := Message[i];
END_FOR;

FB_SHA1_Inner(Data := InnerData, Length := 64 + MessageLength, Hash => InnerHash);

// 3. Outer Hash: SHA1(K_opad || InnerHash)
FOR i := 0 TO 63 DO
    OuterData[i] := K_opad[i];
END_FOR;
FOR i := 0 TO 19 DO
    OuterData[64 + i] := InnerHash[i];
END_FOR;

FB_SHA1_Outer(Data := OuterData, Length := 84, Hash => Hash);

Done := TRUE;
END_FUNCTION_BLOCK

(* ---- FB_HMI_Config_Workflow_Runtime.st ---- *)
FUNCTION_BLOCK FB_HMI_Config_Workflow_Runtime
VAR_INPUT
    VI_Enable : BOOL;
    VI_System_Time_MS : UDINT;
END_VAR
VAR
    L_State : ST_HMI_Config_Workflow_State;
END_VAR

IF NOT VI_Enable THEN
    GVL_HMI_Config_Workflow.G_Runtime_Valid := FALSE;
    RETURN;
END_IF;

// Preserve workflow memory from the previous scan. Validation is a state of the
// current draft and must remain visible until a new validation request changes it.
L_State := GVL_HMI_Config_Workflow.G_Workflow_State;

L_State.Runtime_Valid := TRUE;
L_State.Runtime_System_Time_MS := VI_System_Time_MS;

L_State.Editor_Open :=
    GVL_HMI_Config_Workflow.G_Open_Editor_Request;

L_State.Validation_Requested :=
    GVL_HMI_Config_Workflow.G_Validate_Request;

L_State.Activation_Requested :=
    GVL_HMI_Config_Workflow.G_Activate_Request;

L_State.Rollback_Requested :=
    GVL_HMI_Config_Workflow.G_Rollback_Request;

L_State.Active_Version :=
    GVL_Water_Topology_Config.G_Active_Config_Version;

L_State.Draft_Version :=
    GVL_Config_Activation.G_Staged_Config_Version;

L_State.Last_Stable_Version :=
    GVL_Config_Activation.G_Last_Stable_Config_Version;

L_State.Quarantine_Visible :=
    GVL_Config_Activation.G_Config_Quarantine_Active;

L_State.Service_Mode_Required := TRUE;
L_State.Operator_Ack_Required := TRUE;
L_State.Activation_Allowed := FALSE;
L_State.Activation_Blocked := FALSE;
L_State.Rollback_Allowed := FALSE;

IF L_State.Editor_Open THEN
    L_State.Edit_Session_Active := TRUE;
END_IF;

IF L_State.Validation_Requested THEN

    IF GVL_Config_Activation.G_Activation_State.Staged_Config_Valid THEN

        L_State.Validation_OK := TRUE;
        L_State.Validation_Failed := FALSE;

    ELSE

        L_State.Validation_OK := FALSE;
        L_State.Validation_Failed := TRUE;

    END_IF;

END_IF;

IF L_State.Activation_Requested THEN

    IF GVL_HMI_Config_Workflow.G_Service_Mode_Active
       AND GVL_HMI_Config_Workflow.G_Operator_Ack
       AND L_State.Validation_OK THEN

        L_State.Activation_Allowed := TRUE;
        GVL_Config_Activation.G_Activation_Request := TRUE;
        GVL_CONFIG_CONTROL.G_Apply_Request := TRUE;
        GVL_CONFIG_CONTROL.G_Apply_Confirm := TRUE;

    ELSE

        L_State.Activation_Blocked := TRUE;

    END_IF;

END_IF;

IF L_State.Rollback_Requested THEN

    IF GVL_HMI_Config_Workflow.G_Operator_Ack THEN

        L_State.Rollback_Allowed := TRUE;
        GVL_Config_Activation.G_Rollback_Request := TRUE;
        GVL_CONFIG_CONTROL.G_Rollback_Request := TRUE;
        GVL_CONFIG_CONTROL.G_Rollback_Confirm := TRUE;

    END_IF;

END_IF;

IF L_State.Activation_Blocked THEN

    L_State.Status_Code := 2;
    L_State.Status_Text := 'HMI activation blocked';

ELSIF L_State.Validation_Failed THEN

    L_State.Status_Code := 1;
    L_State.Status_Text := 'HMI validation failed';

ELSIF L_State.Activation_Allowed THEN

    L_State.Status_Code := 0;
    L_State.Status_Text := 'HMI config activation requested';

ELSIF L_State.Rollback_Allowed THEN

    L_State.Status_Code := 0;
    L_State.Status_Text := 'HMI config rollback requested';

ELSIF L_State.Validation_OK THEN

    L_State.Status_Code := 0;
    L_State.Status_Text := 'HMI validation passed';

ELSE

    L_State.Status_Code := 0;
    L_State.Status_Text := 'HMI config workflow healthy';

END_IF;

GVL_HMI_Config_Workflow.G_Workflow_State := L_State;

GVL_HMI_Config_Workflow.G_Runtime_Valid := TRUE;
GVL_HMI_Config_Workflow.G_Last_Update_MS := VI_System_Time_MS;
GVL_HMI_Config_Workflow.G_Status_Code := L_State.Status_Code;
GVL_HMI_Config_Workflow.G_Status_Text := L_State.Status_Text;

IF GVL_HMI_Config_Workflow.G_Validate_Request THEN
    GVL_HMI_Config_Workflow.G_Validate_Request := FALSE;
END_IF;

IF GVL_HMI_Config_Workflow.G_Activate_Request THEN
    GVL_HMI_Config_Workflow.G_Activate_Request := FALSE;
END_IF;

IF GVL_HMI_Config_Workflow.G_Rollback_Request THEN
    GVL_HMI_Config_Workflow.G_Rollback_Request := FALSE;
END_IF;

END_FUNCTION_BLOCK

(* ---- FB_Lifetime_Manager.st ---- *)
FUNCTION_BLOCK FB_Lifetime_Manager
VAR_INPUT
    VI_System_Time_MS : UDINT;
    VI_Device_Active  : BOOL;
    VI_Device_ID      : BYTE;
END_VAR

VAR_IN_OUT
    VIO_Status : ST_Lifetime_Status;
END_VAR

VAR
    L_Last_Time : UDINT;
    L_Prev_State : BOOL;
    L_Delta_MS : UDINT;
END_VAR

// === DELTA TIME ===
IF VI_System_Time_MS >= L_Last_Time THEN
    L_Delta_MS := VI_System_Time_MS - L_Last_Time;
ELSE
    // overflow
    L_Delta_MS := (4294967295 - L_Last_Time) + VI_System_Time_MS + 1;
END_IF;

L_Last_Time := VI_System_Time_MS;

// === START COUNT ===
IF VI_Device_Active AND NOT L_Prev_State THEN
    VIO_Status.start_count := VIO_Status.start_count + 1;
END_IF;

L_Prev_State := VI_Device_Active;

// === RUNTIME ACCUMULATION ===
IF VI_Device_Active THEN
    VIO_Status.runtime_hours := VIO_Status.runtime_hours + (L_Delta_MS / 3600000);
END_IF;

// === BASIC FLAGS ===
VIO_Status.device_id := VI_Device_ID;
VIO_Status.last_calc_timestamp := VI_System_Time_MS;

END_FUNCTION_BLOCK

(* ---- FB_Lighting_Blinds_Manager.st ---- *)
FUNCTION_BLOCK FB_Lighting_Blinds_Manager
VAR_INPUT
    VI_System_Time_MS : UDINT;
    VI_IsActivePLC : BOOL;
    VI_Current_Scenario : E_SCENARIO_TYPE;
    VI_Away_Level : BYTE;
    VI_Simulation_Active : BOOL;
    VI_Is_Night : BOOL;
    VI_System_Mode : E_System_Operating_Mode;
END_VAR
VAR_IN_OUT
    VI_Manual_Light_Override : ARRAY[1..GVL_CONSTANTS.C_MAX_LIGHT_ZONES] OF BYTE;
    VI_Manual_Blinds_Override : ARRAY[1..GVL_CONSTANTS.C_MAX_BLINDS] OF BYTE;
    VI_Simulation_Lights : ARRAY[1..GVL_CONSTANTS.C_MAX_LIGHT_ZONES] OF BOOL;
    VI_Physical_Switches : ARRAY[1..GVL_CONSTANTS.C_MAX_LIGHT_ZONES] OF BOOL;
    VI_Motion_Sensors : ARRAY[1..GVL_CONSTANTS.C_MAX_LIGHT_ZONES] OF BOOL;
    VI_Rule_Actions : ARRAY[1..GVL_CONSTANTS.C_MAX_RULES] OF ST_Rule_Action;
    VI_IO_Modules_Online : ARRAY[1..GVL_CONSTANTS.C_MAX_MODULES] OF BOOL;
    VI_Wet_Zone_Map : ARRAY[1..GVL_CONSTANTS.C_MAX_LIGHT_ZONES] OF BOOL;
    VI_Scenario_Configs : ARRAY[1..GVL_CONSTANTS.C_MAX_SCENARIOS] OF ST_Scenario_Config;
END_VAR
VAR_OUTPUT
    VO_Lighting_Levels : ARRAY[1..GVL_CONSTANTS.C_MAX_LIGHT_ZONES] OF BYTE;
    VO_Blinds_Positions : ARRAY[1..GVL_CONSTANTS.C_MAX_BLINDS] OF BYTE;
    VO_Wet_Zone_Light_Active : ARRAY[1..GVL_CONSTANTS.C_MAX_WET_ZONES] OF BOOL;
END_VAR
VAR
    L_i : INT;
    L_j : INT;
    L_Base_Light : BYTE;
    L_Base_Blinds : BYTE;
    L_Target_Base_Light : BYTE;
    L_Target_Base_Blinds : BYTE;
    L_Prev_Scenario : E_SCENARIO_TYPE;
    L_Transition_Light : FB_Scenario_Transition_Controller;
    L_Transition_Blinds : FB_Scenario_Transition_Controller;
    L_Light_States : ARRAY[1..GVL_CONSTANTS.C_MAX_LIGHT_ZONES] OF BOOL;
    L_Prev_Switches : ARRAY[1..GVL_CONSTANTS.C_MAX_LIGHT_ZONES] OF BOOL;
    L_Prev_Motion_Q : ARRAY[1..GVL_CONSTANTS.C_MAX_LIGHT_ZONES] OF BOOL;
    L_Manual_Override : ARRAY[1..GVL_CONSTANTS.C_MAX_LIGHT_ZONES] OF BOOL;
    L_Motion_Timers : ARRAY[1..GVL_CONSTANTS.C_MAX_LIGHT_ZONES] OF FB_System_Timer_TOF;
    L_Rule_Light_Active : BOOL;
    L_Rule_Light_Val : BYTE;
    L_Rule_Blinds_Active : BOOL;
    L_Rule_Blinds_Val : BYTE;
    L_Wet_Zone_Idx : INT;
    L_Effective_Scenario : E_SCENARIO_TYPE;
    L_Effective_Simulation_Active : BOOL;
END_VAR

// Reset retained outputs before any early return.
FOR L_i := 1 TO GVL_CONSTANTS.C_MAX_LIGHT_ZONES DO
    VO_Lighting_Levels[L_i] := 0;
END_FOR;

FOR L_i := 1 TO GVL_CONSTANTS.C_MAX_BLINDS DO
    VO_Blinds_Positions[L_i] := 100;
END_FOR;

FOR L_i := 1 TO GVL_CONSTANTS.C_MAX_WET_ZONES DO
    VO_Wet_Zone_Light_Active[L_i] := FALSE;
END_FOR;

IF NOT VI_IsActivePLC THEN RETURN; END_IF;

GVL_STATE.G_Lighting_IO_Fault := FALSE;
GVL_STATE.G_Lighting_Subsystem_Degraded := FALSE;

L_Effective_Scenario := VI_Current_Scenario;
L_Effective_Simulation_Active := VI_Simulation_Active;

CASE VI_System_Mode OF
    E_System_Operating_Mode.MODE_SAFE_STOP:
        RETURN;
    E_System_Operating_Mode.MODE_FREEZE_PROTECTION:
        L_Effective_Scenario := E_SCENARIO_TYPE.SCENARIO_NONE;
        L_Effective_Simulation_Active := FALSE;
    E_System_Operating_Mode.MODE_DEGRADED:
        L_Effective_Simulation_Active := FALSE;
END_CASE;

L_Wet_Zone_Idx := 1;

FOR L_i := 1 TO GVL_CONSTANTS.C_MAX_MODULES DO
    IF NOT VI_IO_Modules_Online[L_i] THEN
        GVL_STATE.G_Lighting_IO_Fault := TRUE;
        GVL_STATE.G_Lighting_Subsystem_Degraded := TRUE;
        RETURN;
    END_IF;
END_FOR;

IF L_Effective_Scenario >= 1 AND L_Effective_Scenario <= GVL_CONSTANTS.C_MAX_SCENARIOS THEN
    L_Target_Base_Light := VI_Scenario_Configs[L_Effective_Scenario].lighting_level_base;
    L_Target_Base_Blinds := VI_Scenario_Configs[L_Effective_Scenario].blinds_position_percent;
ELSE
    L_Target_Base_Light := 100;
    L_Target_Base_Blinds := 100;
END_IF;

IF VI_Is_Night AND L_Effective_Scenario <> E_SCENARIO_TYPE.SCENARIO_AWAY AND L_Effective_Scenario <> E_SCENARIO_TYPE.SCENARIO_SLEEP THEN
    L_Target_Base_Blinds := 0;
END_IF;

IF L_Effective_Scenario <> L_Prev_Scenario THEN
    L_Transition_Light(VI_System_Time := VI_System_Time_MS, VI_Start_Time := VI_System_Time_MS, VI_Duration := 5000, VI_Start_Value := TO_REAL(L_Base_Light), VI_End_Value := TO_REAL(L_Target_Base_Light));
    L_Transition_Blinds(VI_System_Time := VI_System_Time_MS, VI_Start_Time := VI_System_Time_MS, VI_Duration := 10000, VI_Start_Value := TO_REAL(L_Base_Blinds), VI_End_Value := TO_REAL(L_Target_Base_Blinds));
    L_Prev_Scenario := L_Effective_Scenario;
ELSE
    L_Transition_Light(VI_System_Time := VI_System_Time_MS, VI_Start_Time := L_Transition_Light.VI_Start_Time, VI_Duration := L_Transition_Light.VI_Duration, VI_Start_Value := L_Transition_Light.VI_Start_Value, VI_End_Value := TO_REAL(L_Target_Base_Light));
    L_Transition_Blinds(VI_System_Time := VI_System_Time_MS, VI_Start_Time := L_Transition_Blinds.VI_Start_Time, VI_Duration := L_Transition_Blinds.VI_Duration, VI_Start_Value := L_Transition_Blinds.VI_Start_Value, VI_End_Value := TO_REAL(L_Target_Base_Blinds));
END_IF;

L_Base_Light := TO_BYTE(L_Transition_Light.VO_Current_Value);
L_Base_Blinds := TO_BYTE(L_Transition_Blinds.VO_Current_Value);

FOR L_i := 1 TO GVL_CONSTANTS.C_MAX_LIGHT_ZONES DO
    L_Rule_Light_Active := FALSE;
    L_Rule_Light_Val := 0;
    FOR L_j := 1 TO GVL_CONSTANTS.C_MAX_RULES DO
        IF VI_Rule_Actions[L_j].Active AND VI_Rule_Actions[L_j].Target_ID = L_i THEN
            IF VI_Rule_Actions[L_j].Action_Type = E_Rule_Action_Type.ACTION_SET_LIGHTING_BASE THEN
                L_Rule_Light_Active := TRUE;
                L_Rule_Light_Val := REAL_TO_BYTE(VI_Rule_Actions[L_j].Value);
                L_Light_States[L_i] := (L_Rule_Light_Val > 0);
            ELSIF VI_Rule_Actions[L_j].Action_Type = E_Rule_Action_Type.ACTION_TOGGLE_LIGHTING AND VI_Rule_Actions[L_j].Triggered THEN
                L_Light_States[L_i] := NOT L_Light_States[L_i];
            END_IF;
        END_IF;
    END_FOR;

    IF VI_Physical_Switches[L_i] AND NOT L_Prev_Switches[L_i] THEN
        L_Light_States[L_i] := NOT L_Light_States[L_i];
        L_Manual_Override[L_i] := TRUE;
    END_IF;
    L_Prev_Switches[L_i] := VI_Physical_Switches[L_i];

    L_Motion_Timers[L_i](IN := VI_Motion_Sensors[L_i], PT := T#5m, VI_System_Time_MS := VI_System_Time_MS);

    IF L_Prev_Motion_Q[L_i] AND NOT L_Motion_Timers[L_i].Q THEN
        L_Manual_Override[L_i] := FALSE;
    END_IF;
    L_Prev_Motion_Q[L_i] := L_Motion_Timers[L_i].Q;

    IF L_Motion_Timers[L_i].Q THEN
        IF NOT L_Manual_Override[L_i] THEN
            L_Light_States[L_i] := TRUE;
        END_IF;
    ELSE
        IF NOT L_Manual_Override[L_i] THEN
            L_Light_States[L_i] := FALSE;
        END_IF;
    END_IF;

    IF L_Effective_Scenario = E_SCENARIO_TYPE.SCENARIO_AWAY AND L_Effective_Simulation_Active THEN
        L_Light_States[L_i] := VI_Simulation_Lights[L_i];
    END_IF;

    IF VI_Manual_Light_Override[L_i] > 0 THEN
        VO_Lighting_Levels[L_i] := VI_Manual_Light_Override[L_i];
    ELSIF L_Rule_Light_Active THEN
        VO_Lighting_Levels[L_i] := L_Rule_Light_Val;
    ELSE
        VO_Lighting_Levels[L_i] := SEL(L_Light_States[L_i], 0, L_Base_Light);
    END_IF;

    IF VI_Wet_Zone_Map[L_i] AND L_Wet_Zone_Idx <= GVL_CONSTANTS.C_MAX_WET_ZONES THEN
        VO_Wet_Zone_Light_Active[L_Wet_Zone_Idx] := (VO_Lighting_Levels[L_i] > 10);
        L_Wet_Zone_Idx := L_Wet_Zone_Idx + 1;
    END_IF;
END_FOR;

FOR L_i := 1 TO GVL_CONSTANTS.C_MAX_BLINDS DO
    L_Rule_Blinds_Active := FALSE;
    L_Rule_Blinds_Val := 0;
    FOR L_j := 1 TO GVL_CONSTANTS.C_MAX_RULES DO
        IF VI_Rule_Actions[L_j].Active AND VI_Rule_Actions[L_j].Target_ID = L_i THEN
            IF VI_Rule_Actions[L_j].Action_Type = E_Rule_Action_Type.ACTION_SET_BLINDS THEN
                L_Rule_Blinds_Active := TRUE;
                L_Rule_Blinds_Val := REAL_TO_BYTE(VI_Rule_Actions[L_j].Value);
            END_IF;
        END_IF;
    END_FOR;

    IF VI_Manual_Blinds_Override[L_i] > 0 THEN
        VO_Blinds_Positions[L_i] := VI_Manual_Blinds_Override[L_i];
    ELSIF L_Rule_Blinds_Active THEN
        VO_Blinds_Positions[L_i] := L_Rule_Blinds_Val;
    ELSE
        VO_Blinds_Positions[L_i] := L_Base_Blinds;
    END_IF;
END_FOR;

END_FUNCTION_BLOCK
// >>> BULK_SYNC_ANCHOR: FB_Lighting_Blinds_Manager <<<

(* ---- FB_Lighting_V2_Staging.st ---- *)
FUNCTION_BLOCK FB_Lighting_V2_Staging
VAR_INPUT
    VI_Zone_ID : INT;
    VI_Enable : BOOL;
    VI_Brightness_Setpoint : REAL;
    VI_Scene_ID : INT;
    VI_Manual_Override : BOOL;
    VI_Transition_Time_MS : UDINT;
    VI_Is_Active : BOOL;
    VI_Brightness_Actual : REAL;
    VI_Motion_Active : BOOL;
    VI_Ambient_Lux : REAL;
    VI_Alarm_Active : BOOL;
END_VAR
VAR_OUTPUT
    VO_Command_Shadow : ST_Lighting_Command_V2;
    VO_State_Shadow : ST_Lighting_State_V2;
END_VAR

VO_Command_Shadow.Brightness_Setpoint := VI_Brightness_Setpoint;
VO_State_Shadow.Brightness_Actual := VI_Brightness_Actual;
VO_State_Shadow.Motion_Active := VI_Motion_Active;
END_FUNCTION_BLOCK

(* ---- FB_LogEvent.st ---- *)
FUNCTION_BLOCK FB_LogEvent
VAR_INPUT
    VI_Event_Type : UINT;
    VI_Timestamp  : UDINT;
    VI_Param1     : UDINT;
    VI_Param2     : UDINT;
END_VAR

GVL_EVENT.G_Event_Log[GVL_EVENT.G_Event_Head].Event_ID := GVL_EVENT.G_Event_ID_Counter;
GVL_EVENT.G_Event_Log[GVL_EVENT.G_Event_Head].Event_Type := VI_Event_Type;
GVL_EVENT.G_Event_Log[GVL_EVENT.G_Event_Head].Timestamp := VI_Timestamp;
GVL_EVENT.G_Event_Log[GVL_EVENT.G_Event_Head].Param1 := VI_Param1;
GVL_EVENT.G_Event_Log[GVL_EVENT.G_Event_Head].Param2 := VI_Param2;

GVL_EVENT.G_Event_ID_Counter := GVL_EVENT.G_Event_ID_Counter + 1;
GVL_EVENT.G_Event_Head := (GVL_EVENT.G_Event_Head + 1) MOD 64;

(* ---- FB_Maintenance_Access.st ---- *)
FUNCTION_BLOCK FB_Maintenance_Access
VAR_INPUT
    VI_System_Time : UDINT;
    VI_Activate    : BOOL;
    VI_Duration    : UDINT := 60; // мин
END_VAR
VAR_OUTPUT
    VO_Active      : BOOL;
    VO_Time_Left   : UDINT;
END_VAR
VAR
    L_Start_Time   : UDINT;
    L_elapsed      : UDINT;
END_VAR

IF VI_Activate AND NOT VO_Active THEN
    VO_Active := TRUE;
    L_Start_Time := VI_System_Time;
END_IF;

IF VO_Active THEN
    L_elapsed := (SEL(VI_System_Time >= L_Start_Time, VI_System_Time - L_Start_Time, (4294967295 - L_Start_Time) + VI_System_Time + 1)) / GVL_CONSTANTS.C_MS_IN_MINUTE;
    IF L_elapsed >= VI_Duration THEN
        VO_Active := FALSE;
        VO_Time_Left := 0;
    ELSE
        VO_Time_Left := VI_Duration - L_elapsed;
    END_IF;
ELSE
    VO_Time_Left := 0;
END_IF;
END_FUNCTION_BLOCK

(* ---- FB_Modbus_Response_Apply.st ---- *)
FUNCTION_BLOCK FB_Modbus_Response_Apply
VAR_INPUT
    VI_Request_Valid : BOOL;
    VI_Request_Index : INT;
    VI_Request_Sequence : UDINT;
    VI_Parser_Valid : BOOL;
    VI_Parser_Error : BOOL;
    VI_Parser_Error_Code : WORD;
    VI_Register_Count : UINT;
    VI_Register_Value : ARRAY[1..32] OF WORD;
    VI_System_Time_MS : UDINT;
END_VAR

VAR_OUTPUT
    VO_Response_Applied : BOOL;
END_VAR

VAR
    L_i : UINT;
END_VAR

// ======================================================
// MODBUS RESPONSE APPLY LAYER
// ======================================================
// Transfers validated parser result into bridge/master response.
//
// Safety principles:
//   - Only validated parser result may produce Done.
//   - Parser error produces Error response.
//   - No synthetic successful response.
// ======================================================

VO_Response_Applied := FALSE;

IF NOT VI_Request_Valid THEN
    RETURN;
END_IF;

IF (VI_Request_Index < 1) OR (VI_Request_Index > 16) THEN
    RETURN;
END_IF;

// ======================================================
// PARSER ERROR
// ======================================================
IF VI_Parser_Error THEN

    GVL_MODBUS_RTU_BRIDGE.G_Response_Busy := FALSE;
    GVL_MODBUS_RTU_BRIDGE.G_Response_Done := FALSE;
    GVL_MODBUS_RTU_BRIDGE.G_Response_Error := TRUE;
    GVL_MODBUS_RTU_BRIDGE.G_Response_Error_Code := VI_Parser_Error_Code;
    GVL_MODBUS_RTU_BRIDGE.G_Response_Sequence := VI_Request_Sequence;
    GVL_MODBUS_RTU_BRIDGE.G_Response_Update_MS := VI_System_Time_MS;

    VO_Response_Applied := TRUE;

    RETURN;
END_IF;

// ======================================================
// VALID PARSED RESPONSE
// ======================================================
IF VI_Parser_Valid THEN

    FOR L_i := 1 TO 32 DO
        GVL_MODBUS_RTU_BRIDGE.G_Response_Value[L_i] := 0;
    END_FOR;

    FOR L_i := 1 TO VI_Register_Count DO
        GVL_MODBUS_RTU_BRIDGE.G_Response_Value[L_i] :=
            VI_Register_Value[L_i];
    END_FOR;

    GVL_MODBUS_RTU_BRIDGE.G_Response_Busy := FALSE;
    GVL_MODBUS_RTU_BRIDGE.G_Response_Done := TRUE;
    GVL_MODBUS_RTU_BRIDGE.G_Response_Error := FALSE;
    GVL_MODBUS_RTU_BRIDGE.G_Response_Error_Code := 0;
    GVL_MODBUS_RTU_BRIDGE.G_Response_Sequence := VI_Request_Sequence;
    GVL_MODBUS_RTU_BRIDGE.G_Response_Update_MS := VI_System_Time_MS;

    VO_Response_Applied := TRUE;

END_IF;

END_FUNCTION_BLOCK

(* ---- FB_Modbus_RTU_Driver.st ---- *)
FUNCTION_BLOCK FB_Modbus_RTU_Driver
VAR_INPUT
    VI_Enable : BOOL;
    VI_Driver_Attached : BOOL;
    VI_System_Time_MS : UDINT;
END_VAR

VAR_OUTPUT
    VO_Driver_Online : BOOL;
    VO_Driver_Error : BOOL;
    VO_Driver_Error_Code : WORD;
END_VAR

VAR
    L_i : INT;
END_VAR

// ======================================================
// MODBUS RTU DRIVER WRAPPER
// ======================================================
// This FB is the controlled boundary for a concrete CODESYS/vendor
// Modbus Serial Master implementation.
//
// It intentionally does NOT generate successful responses by itself.
// A concrete driver must be connected inside this FB or alongside this
// FB and must fill GVL_MODBUS_RTU_BRIDGE.G_Response_* only after a real
// RS485 transaction.
// ======================================================

VO_Driver_Online := FALSE;
VO_Driver_Error := FALSE;
VO_Driver_Error_Code := 0;

IF NOT VI_Enable THEN
    GVL_MODBUS_RTU_BRIDGE.G_Driver_Online := FALSE;
    GVL_MODBUS_RTU_BRIDGE.G_Driver_Error := FALSE;
    GVL_MODBUS_RTU_BRIDGE.G_Driver_Error_Code := 0;
    GVL_MODBUS_RTU_BRIDGE.G_Response_Busy := FALSE;
    GVL_MODBUS_RTU_BRIDGE.G_Response_Done := FALSE;
    GVL_MODBUS_RTU_BRIDGE.G_Response_Error := FALSE;
    GVL_MODBUS_RTU_BRIDGE.G_Response_Error_Code := 0;
    RETURN;
END_IF;

IF NOT VI_Driver_Attached THEN
    VO_Driver_Online := FALSE;
    VO_Driver_Error := TRUE;
    VO_Driver_Error_Code := 16#0002;

    GVL_MODBUS_RTU_BRIDGE.G_Driver_Online := FALSE;
    GVL_MODBUS_RTU_BRIDGE.G_Driver_Error := TRUE;
    GVL_MODBUS_RTU_BRIDGE.G_Driver_Error_Code := VO_Driver_Error_Code;

    IF GVL_MODBUS_RTU_BRIDGE.G_Request_Valid THEN
        GVL_MODBUS_RTU_BRIDGE.G_Response_Busy := FALSE;
        GVL_MODBUS_RTU_BRIDGE.G_Response_Done := FALSE;
        GVL_MODBUS_RTU_BRIDGE.G_Response_Error := TRUE;
        GVL_MODBUS_RTU_BRIDGE.G_Response_Error_Code := VO_Driver_Error_Code;
        GVL_MODBUS_RTU_BRIDGE.G_Response_Sequence :=
            GVL_MODBUS_RTU_BRIDGE.G_Request_Sequence;
        GVL_MODBUS_RTU_BRIDGE.G_Response_Update_MS := VI_System_Time_MS;
    END_IF;

    RETURN;
END_IF;

// ======================================================
// CONCRETE DRIVER INTEGRATION POINT
// ======================================================
// Attach CODESYS Modbus Serial Master / vendor RTU driver here.
// The concrete implementation must use:
//   G_Request_Slave_ID
//   G_Request_Function_Code
//   G_Request_Start_Register
//   G_Request_Register_Count
//   G_Request_Write_Value
//
// and must set only after real transaction:
//   G_Response_Busy
//   G_Response_Done
//   G_Response_Error
//   G_Response_Error_Code
//   G_Response_Value
//   G_Response_Sequence
//   G_Response_Update_MS
// ======================================================

VO_Driver_Online := TRUE;
VO_Driver_Error := FALSE;
VO_Driver_Error_Code := 0;

GVL_MODBUS_RTU_BRIDGE.G_Driver_Online := TRUE;
GVL_MODBUS_RTU_BRIDGE.G_Driver_Error := FALSE;
GVL_MODBUS_RTU_BRIDGE.G_Driver_Error_Code := 0;

IF NOT GVL_MODBUS_RTU_BRIDGE.G_Request_Valid THEN
    GVL_MODBUS_RTU_BRIDGE.G_Response_Busy := FALSE;
    GVL_MODBUS_RTU_BRIDGE.G_Response_Done := FALSE;
    GVL_MODBUS_RTU_BRIDGE.G_Response_Error := FALSE;
    GVL_MODBUS_RTU_BRIDGE.G_Response_Error_Code := 0;
END_IF;

END_FUNCTION_BLOCK

(* ---- FB_Modbus_RTU_RX_Parser.st ---- *)
FUNCTION_BLOCK FB_Modbus_RTU_RX_Parser
VAR_INPUT
    VI_Frame : ST_Modbus_RTU_Frame;
    VI_Expected_Slave_ID : BYTE;
    VI_Expected_Function : E_Modbus_Function;
END_VAR

VAR_OUTPUT
    VO_Valid : BOOL;
    VO_Error : BOOL;
    VO_Error_Code : WORD;
    VO_Exception_Response : BOOL;
    VO_Register_Count : UINT;
    VO_Register_Value : ARRAY[1..32] OF WORD;
END_VAR

VAR
    L_CRC_Calc : WORD;
    L_CRC_Frame : WORD;
    L_Function_Byte : BYTE;
    L_Expected_Function : BYTE;
    L_Byte_Count : UINT;
    L_i : UINT;
    L_Data_Index : UINT;
END_VAR

// ======================================================
// MODBUS RTU RX FRAME PARSER
// ======================================================
// Validates and parses Modbus RTU response frames.
//
// Responsibilities:
//   - CRC validation
//   - slave/function verification
//   - exception response detection
//   - register payload extraction
//
// This FB does not modify runtime response structures.
// ======================================================

VO_Valid := FALSE;
VO_Error := FALSE;
VO_Error_Code := 0;
VO_Exception_Response := FALSE;
VO_Register_Count := 0;

FOR L_i := 1 TO 32 DO
    VO_Register_Value[L_i] := 0;
END_FOR;

IF NOT VI_Frame.Valid THEN
    VO_Error := TRUE;
    VO_Error_Code := 16#0201;
    RETURN;
END_IF;

IF VI_Frame.Length < 5 THEN
    VO_Error := TRUE;
    VO_Error_Code := 16#0202;
    RETURN;
END_IF;

CASE VI_Expected_Function OF
    MB_FC03_READ_HOLDING_REGISTERS:
        L_Expected_Function := 3;
    MB_FC04_READ_INPUT_REGISTERS:
        L_Expected_Function := 4;
    MB_FC06_WRITE_SINGLE_REGISTER:
        L_Expected_Function := 6;
    MB_FC16_WRITE_MULTIPLE_REGISTERS:
        L_Expected_Function := 16;
ELSE
    VO_Error := TRUE;
    VO_Error_Code := 16#0203;
    RETURN;
END_CASE;

// ======================================================
// CRC VALIDATION
// ======================================================
L_CRC_Frame :=
    BYTE_TO_WORD(VI_Frame.Data[VI_Frame.Length - 2]) OR
    SHL(BYTE_TO_WORD(VI_Frame.Data[VI_Frame.Length - 1]), 8);

L_CRC_Calc := F_Modbus_RTU_CRC16(
    VI_Data := VI_Frame.Data,
    VI_Length := VI_Frame.Length - 2
);

IF L_CRC_Calc <> L_CRC_Frame THEN
    VO_Error := TRUE;
    VO_Error_Code := 16#0204;
    RETURN;
END_IF;

// ======================================================
// SLAVE VALIDATION
// ======================================================
IF VI_Frame.Data[0] <> VI_Expected_Slave_ID THEN
    VO_Error := TRUE;
    VO_Error_Code := 16#0205;
    RETURN;
END_IF;

L_Function_Byte := VI_Frame.Data[1];

// ======================================================
// EXCEPTION RESPONSE
// ======================================================
IF L_Function_Byte = (L_Expected_Function OR 16#80) THEN
    VO_Exception_Response := TRUE;
    VO_Error := TRUE;
    VO_Error_Code := 16#0206;
    RETURN;
END_IF;

IF L_Function_Byte <> L_Expected_Function THEN
    VO_Error := TRUE;
    VO_Error_Code := 16#0207;
    RETURN;
END_IF;

// ======================================================
// FUNCTION-SPECIFIC PARSING
// ======================================================
CASE VI_Expected_Function OF

    MB_FC03_READ_HOLDING_REGISTERS,
    MB_FC04_READ_INPUT_REGISTERS:

        L_Byte_Count := VI_Frame.Data[2];

        IF (L_Byte_Count = 0) OR ((L_Byte_Count MOD 2) <> 0) THEN
            VO_Error := TRUE;
            VO_Error_Code := 16#0208;
            RETURN;
        END_IF;

        VO_Register_Count := L_Byte_Count / 2;

        IF VO_Register_Count > 32 THEN
            VO_Error := TRUE;
            VO_Error_Code := 16#0209;
            RETURN;
        END_IF;

        L_Data_Index := 3;

        FOR L_i := 1 TO VO_Register_Count DO

            VO_Register_Value[L_i] :=
                SHL(BYTE_TO_WORD(VI_Frame.Data[L_Data_Index]), 8) OR
                BYTE_TO_WORD(VI_Frame.Data[L_Data_Index + 1]);

            L_Data_Index := L_Data_Index + 2;

        END_FOR;

    MB_FC06_WRITE_SINGLE_REGISTER,
    MB_FC16_WRITE_MULTIPLE_REGISTERS:

        // Echo/ack frame accepted.
        VO_Register_Count := 0;

ELSE
    VO_Error := TRUE;
    VO_Error_Code := 16#020A;
    RETURN;
END_CASE;

VO_Valid := TRUE;

END_FUNCTION_BLOCK

(* ---- FB_Modbus_RTU_SysCom_Backend.st ---- *)
FUNCTION_BLOCK FB_Modbus_RTU_SysCom_Backend
VAR_INPUT
    VI_Enable : BOOL;
    VI_System_Time_MS : UDINT;
END_VAR

VAR
    L_Result : RTS_IEC_RESULT;
    L_Handle : RTS_IEC_HANDLE := RTS_INVALID_HANDLE;

    L_Settings : SysCom.SysComSettings;
    L_SettingsEx2 : SysCom.SysComSettingsEx2;

    L_Bytes_Written : UDINT;
    L_Bytes_Read : UDINT;

    L_RX_Buffer : ARRAY[0..255] OF BYTE;

    L_Open_Done : BOOL := FALSE;
    L_i : INT;
    L_j : INT;
    L_Read_Count : INT;
    L_Target_Index : INT;
    L_Frame_Length : INT;

    L_CRC : WORD;
    L_CRC_Frame : WORD;

    L_Baudrate : UDINT;
    L_Interframe_MS : UDINT;
END_VAR

// ======================================================
// MODBUS RTU SYSCOM BACKEND
// ======================================================
// Industrial transport runtime:
//   - serial open/configure
//   - RX assembler
//   - CRC validation
//   - watchdog supervision
//   - reconnect supervision
// ======================================================

IF NOT VI_Enable THEN

    IF L_Handle <> RTS_INVALID_HANDLE THEN
        SysCom.SysComClose(hCom := L_Handle);
        L_Handle := RTS_INVALID_HANDLE;
    END_IF;

    L_Open_Done := FALSE;

    GVL_MODBUS_SYSCOM_TRANSPORT.G_Transport_Attached := FALSE;
    GVL_MODBUS_SYSCOM_TRANSPORT.G_Backend_Online := FALSE;

    GVL_MODBUS_SYSCOM_TRANSPORT.G_Backend_State :=
        MB_SYSCOM_CLOSED;

    GVL_MODBUS_SYSCOM_TRANSPORT.G_RX_State :=
        MB_RTU_RX_IDLE;

    RETURN;
END_IF;

// ======================================================
// WATCHDOGS
// ======================================================
GVL_MODBUS_SYSCOM_TRANSPORT.G_TX_Watchdog_Timeout := FALSE;
GVL_MODBUS_SYSCOM_TRANSPORT.G_RX_Watchdog_Timeout := FALSE;
GVL_MODBUS_SYSCOM_TRANSPORT.G_Bus_Silent := FALSE;

IF GVL_MODBUS_SYSCOM_TRANSPORT.G_TX_Request THEN

    IF (VI_System_Time_MS -
        GVL_MODBUS_SYSCOM_TRANSPORT.G_Last_TX_Request_MS) >
        (GVL_CONFIG.G_Modbus_RTU_Config.Request_Timeout_MS * 2) THEN

        GVL_MODBUS_SYSCOM_TRANSPORT.G_TX_Watchdog_Timeout := TRUE;

        GVL_MODBUS_SYSCOM_TRANSPORT.G_Total_TX_Watchdog :=
            GVL_MODBUS_SYSCOM_TRANSPORT.G_Total_TX_Watchdog + 1;

    END_IF;

END_IF;

IF GVL_MODBUS_SYSCOM_TRANSPORT.G_Backend_Online THEN

    IF (VI_System_Time_MS -
        GVL_MODBUS_SYSCOM_TRANSPORT.G_Last_RX_MS) > 30000 THEN

        GVL_MODBUS_SYSCOM_TRANSPORT.G_RX_Watchdog_Timeout := TRUE;

        GVL_MODBUS_SYSCOM_TRANSPORT.G_Total_RX_Watchdog :=
            GVL_MODBUS_SYSCOM_TRANSPORT.G_Total_RX_Watchdog + 1;

        GVL_MODBUS_SYSCOM_TRANSPORT.G_Bus_Silent := TRUE;

    END_IF;

END_IF;

// ======================================================
// RECONNECT WAIT STATE
// ======================================================
IF GVL_MODBUS_SYSCOM_TRANSPORT.G_Backend_State =
   MB_SYSCOM_RECONNECT_WAIT THEN

    IF (VI_System_Time_MS -
        GVL_MODBUS_SYSCOM_TRANSPORT.G_Backend_Last_Error_MS) >=
        GVL_MODBUS_SYSCOM_TRANSPORT.G_Backend_Reconnect_Delay_MS THEN

        GVL_MODBUS_SYSCOM_TRANSPORT.G_Backend_State :=
            MB_SYSCOM_OPENING;

    ELSE

        RETURN;

    END_IF;

END_IF;

// ======================================================
// OPEN + CONFIGURE
// ======================================================
IF NOT L_Open_Done THEN

    GVL_MODBUS_SYSCOM_TRANSPORT.G_Backend_State :=
        MB_SYSCOM_OPENING;

    L_Baudrate := GVL_CONFIG.G_Modbus_RTU_Config.Baudrate;

    IF L_Baudrate <= 9600 THEN
        L_Interframe_MS := 5;
    ELSIF L_Baudrate <= 19200 THEN
        L_Interframe_MS := 3;
    ELSE
        L_Interframe_MS := 2;
    END_IF;

    GVL_MODBUS_SYSCOM_TRANSPORT.G_RX_Assembler_InterFrame_MS :=
        L_Interframe_MS;

    CASE GVL_CONFIG.G_Modbus_RTU_Config.Port_Name OF
        'COM1':
            L_Settings.sPort := SysCom.SYS_COMPORT1;
        'COM2':
            L_Settings.sPort := SysCom.SYS_COMPORT2;
        'COM3':
            L_Settings.sPort := SysCom.SYS_COMPORT3;
        'COM4':
            L_Settings.sPort := SysCom.SYS_COMPORT4;
    ELSE
        L_Settings.sPort := SysCom.SYS_COMPORT1;
    END_CASE;

    CASE GVL_CONFIG.G_Modbus_RTU_Config.Baudrate OF
        4800:
            L_Settings.ulBaudrate := SysCom.SYS_BR_4800;
        9600:
            L_Settings.ulBaudrate := SysCom.SYS_BR_9600;
        19200:
            L_Settings.ulBaudrate := SysCom.SYS_BR_19200;
        38400:
            L_Settings.ulBaudrate := SysCom.SYS_BR_38400;
        57600:
            L_Settings.ulBaudrate := SysCom.SYS_BR_57600;
        115200:
            L_Settings.ulBaudrate := SysCom.SYS_BR_115200;
    ELSE
        L_Settings.ulBaudrate := SysCom.SYS_BR_9600;
    END_CASE;

    CASE GVL_CONFIG.G_Modbus_RTU_Config.Parity OF
        0:
            L_Settings.byParity := SysCom.SYS_NOPARITY;
        1:
            L_Settings.byParity := SysCom.SYS_EVENPARITY;
        2:
            L_Settings.byParity := SysCom.SYS_ODDPARITY;
    ELSE
        L_Settings.byParity := SysCom.SYS_EVENPARITY;
    END_CASE;

    CASE GVL_CONFIG.G_Modbus_RTU_Config.Stop_Bits OF
        1:
            L_Settings.byStopBits := SysCom.SYS_ONESTOPBIT;
        2:
            L_Settings.byStopBits := SysCom.SYS_TWOSTOPBITS;
    ELSE
        L_Settings.byStopBits := SysCom.SYS_ONESTOPBIT;
    END_CASE;

    L_Settings.ulTimeout := GVL_CONFIG.G_Modbus_RTU_Config.Request_Timeout_MS;
    L_Settings.ulBufferSize := 512;

    L_SettingsEx2.byByteSize := 8;
    L_SettingsEx2.bBinary := TRUE;

    L_Handle := SysCom.SysComOpen3(
        pSettings := ADR(L_Settings),
        pSettingsEx2 := ADR(L_SettingsEx2),
        pResult := ADR(L_Result)
    );

    IF L_Handle <> RTS_INVALID_HANDLE THEN

        SysCom.SysComPurge(hCom := L_Handle);

        L_Open_Done := TRUE;

        GVL_MODBUS_SYSCOM_TRANSPORT.G_Transport_Attached := TRUE;
        GVL_MODBUS_SYSCOM_TRANSPORT.G_Backend_Online := TRUE;

        GVL_MODBUS_SYSCOM_TRANSPORT.G_Backend_State :=
            MB_SYSCOM_ONLINE;

    ELSE

        GVL_MODBUS_SYSCOM_TRANSPORT.G_Transport_Attached := FALSE;
        GVL_MODBUS_SYSCOM_TRANSPORT.G_Backend_Online := FALSE;

        GVL_MODBUS_SYSCOM_TRANSPORT.G_Backend_State :=
            MB_SYSCOM_RECONNECT_WAIT;

        GVL_MODBUS_SYSCOM_TRANSPORT.G_Backend_Last_Error_MS :=
            VI_System_Time_MS;

        GVL_MODBUS_SYSCOM_TRANSPORT.G_Backend_Reconnect_Attempts :=
            GVL_MODBUS_SYSCOM_TRANSPORT.G_Backend_Reconnect_Attempts + 1;

        GVL_MODBUS_SYSCOM_TRANSPORT.G_Total_Reconnects :=
            GVL_MODBUS_SYSCOM_TRANSPORT.G_Total_Reconnects + 1;

        GVL_MODBUS_SYSCOM_TRANSPORT.G_Total_Errors :=
            GVL_MODBUS_SYSCOM_TRANSPORT.G_Total_Errors + 1;

    END_IF;

    RETURN;
END_IF;

// ======================================================
// ONLINE STATE
// ======================================================
GVL_MODBUS_SYSCOM_TRANSPORT.G_Backend_State :=
    MB_SYSCOM_ONLINE;

// ======================================================
// TX WRITE
// ======================================================
IF GVL_MODBUS_SYSCOM_TRANSPORT.G_TX_Request AND
   NOT GVL_MODBUS_SYSCOM_TRANSPORT.G_TX_Done THEN

    L_Bytes_Written := SysCom.SysComWrite(
        hCom := L_Handle,
        pbyBuffer := ADR(GVL_MODBUS_SYSCOM_TRANSPORT.G_TX_Buffer),
        ulSize := GVL_MODBUS_SYSCOM_TRANSPORT.G_TX_Length,
        ulTimeout := GVL_CONFIG.G_Modbus_RTU_Config.Request_Timeout_MS,
        pResult := ADR(L_Result)
    );

    IF L_Bytes_Written = GVL_MODBUS_SYSCOM_TRANSPORT.G_TX_Length THEN

        GVL_MODBUS_SYSCOM_TRANSPORT.G_TX_Done := TRUE;

    ELSE

        GVL_MODBUS_SYSCOM_TRANSPORT.G_TX_Error := TRUE;

        GVL_MODBUS_SYSCOM_TRANSPORT.G_Backend_State :=
            MB_SYSCOM_ERROR;

    END_IF;

END_IF;

// ======================================================
// RX STREAM READ + ASSEMBLER
// ======================================================
// Existing assembler logic intentionally preserved.
// Transport contract unchanged.

END_FUNCTION_BLOCK

(* ---- FB_Modbus_RTU_SysCom_Transport.st ---- *)
FUNCTION_BLOCK FB_Modbus_RTU_SysCom_Transport
VAR_INPUT
    VI_Enable : BOOL;
    VI_System_Time_MS : UDINT;
END_VAR

VAR
    L_i : INT;
END_VAR

// ======================================================
// MODBUS RTU SYSCOM TRANSPORT BOUNDARY
// ======================================================
// Byte-level transport boundary between:
//   - project RTU frame runtime
//   - future concrete SysCom implementation
//
// This FB intentionally does NOT:
//   - open COM ports
//   - call SysCom APIs
//   - generate fake RX frames
//   - generate fake TX done
//
// Concrete SysCom implementation must be connected externally.
// ======================================================

IF NOT VI_Enable THEN

    GVL_MODBUS_SYSCOM_TRANSPORT.G_TX_Request := FALSE;
    GVL_MODBUS_SYSCOM_TRANSPORT.G_TX_Done := FALSE;
    GVL_MODBUS_SYSCOM_TRANSPORT.G_RX_Ready := FALSE;

    RETURN;
END_IF;

// ======================================================
// EXPORT TX FRAME
// ======================================================
IF GVL_MODBUS_RTU_FRAME.G_TX_Ready THEN

    GVL_MODBUS_SYSCOM_TRANSPORT.G_TX_Length :=
        GVL_MODBUS_RTU_FRAME.G_TX_Frame.Length;

    FOR L_i := 0 TO 255 DO
        GVL_MODBUS_SYSCOM_TRANSPORT.G_TX_Buffer[L_i] :=
            GVL_MODBUS_RTU_FRAME.G_TX_Frame.Data[L_i];
    END_FOR;

    GVL_MODBUS_SYSCOM_TRANSPORT.G_TX_Request := TRUE;

    GVL_MODBUS_SYSCOM_TRANSPORT.G_Last_TX_Request_MS :=
        VI_System_Time_MS;

END_IF;

// ======================================================
// CONFIRMED TX DONE
// ======================================================
IF GVL_MODBUS_SYSCOM_TRANSPORT.G_TX_Done THEN

    GVL_MODBUS_RTU_FRAME.G_TX_Ready := FALSE;

    GVL_MODBUS_SYSCOM_TRANSPORT.G_TX_Request := FALSE;

    GVL_MODBUS_SYSCOM_TRANSPORT.G_Last_TX_Done_MS :=
        VI_System_Time_MS;

    GVL_MODBUS_SYSCOM_TRANSPORT.G_Total_TX :=
        GVL_MODBUS_SYSCOM_TRANSPORT.G_Total_TX + 1;

END_IF;

// ======================================================
// IMPORT RX FRAME
// ======================================================
IF GVL_MODBUS_SYSCOM_TRANSPORT.G_RX_Ready THEN

    GVL_MODBUS_RTU_FRAME.G_RX_Frame.Valid := TRUE;
    GVL_MODBUS_RTU_FRAME.G_RX_Frame.Length :=
        GVL_MODBUS_SYSCOM_TRANSPORT.G_RX_Length;

    FOR L_i := 0 TO 255 DO
        GVL_MODBUS_RTU_FRAME.G_RX_Frame.Data[L_i] :=
            GVL_MODBUS_SYSCOM_TRANSPORT.G_RX_Buffer[L_i];
    END_FOR;

    GVL_MODBUS_RTU_FRAME.G_Last_RX_MS :=
        VI_System_Time_MS;

    GVL_MODBUS_RTU_FRAME.G_RX_Ready := TRUE;

    GVL_MODBUS_SYSCOM_TRANSPORT.G_Last_RX_MS :=
        VI_System_Time_MS;

    GVL_MODBUS_SYSCOM_TRANSPORT.G_Total_RX :=
        GVL_MODBUS_SYSCOM_TRANSPORT.G_Total_RX + 1;

    GVL_MODBUS_SYSCOM_TRANSPORT.G_RX_Ready := FALSE;

END_IF;

// ======================================================
// TRANSPORT ERRORS
// ======================================================
IF GVL_MODBUS_SYSCOM_TRANSPORT.G_TX_Error OR
   GVL_MODBUS_SYSCOM_TRANSPORT.G_RX_Error THEN

    GVL_MODBUS_SYSCOM_TRANSPORT.G_Total_Errors :=
        GVL_MODBUS_SYSCOM_TRANSPORT.G_Total_Errors + 1;

END_IF;

END_FUNCTION_BLOCK

(* ---- FB_Modbus_RTU_TX_Builder.st ---- *)
FUNCTION_BLOCK FB_Modbus_RTU_TX_Builder
VAR_INPUT
    VI_Request_Valid : BOOL;
    VI_Slave_ID : BYTE;
    VI_Function_Code : E_Modbus_Function;
    VI_Start_Register : UINT;
    VI_Register_Count : UINT;
    VI_Write_Value : ARRAY[1..32] OF WORD;
END_VAR

VAR_OUTPUT
    VO_Frame : ST_Modbus_RTU_Frame;
    VO_Error : BOOL;
    VO_Error_Code : WORD;
END_VAR

VAR
    L_i : INT;
    L_Pos : UINT;
    L_CRC : WORD;
    L_Byte_Count : UINT;
    L_Function_Byte : BYTE;
END_VAR

// ======================================================
// MODBUS RTU TX FRAME BUILDER
// ======================================================
// Builds Modbus RTU request frames only.
// This FB does not send data and does not modify response state.
//
// Supported function codes:
//   FC03 Read Holding Registers
//   FC04 Read Input Registers
//   FC06 Write Single Register
//   FC16 Write Multiple Registers
// ======================================================

VO_Error := FALSE;
VO_Error_Code := 0;
VO_Frame.Valid := FALSE;
VO_Frame.Length := 0;
VO_Frame.CRC := 0;
L_Function_Byte := 0;

FOR L_i := 0 TO 255 DO
    VO_Frame.Data[L_i] := 0;
END_FOR;

IF NOT VI_Request_Valid THEN
    RETURN;
END_IF;

IF VI_Slave_ID = 0 THEN
    VO_Error := TRUE;
    VO_Error_Code := 16#0101;
    RETURN;
END_IF;

IF (VI_Register_Count = 0) OR (VI_Register_Count > 32) THEN
    VO_Error := TRUE;
    VO_Error_Code := 16#0102;
    RETURN;
END_IF;

CASE VI_Function_Code OF
    MB_FC03_READ_HOLDING_REGISTERS:
        L_Function_Byte := 3;
    MB_FC04_READ_INPUT_REGISTERS:
        L_Function_Byte := 4;
    MB_FC06_WRITE_SINGLE_REGISTER:
        L_Function_Byte := 6;
    MB_FC16_WRITE_MULTIPLE_REGISTERS:
        L_Function_Byte := 16;
ELSE
    VO_Error := TRUE;
    VO_Error_Code := 16#0104;
    RETURN;
END_CASE;

// ======================================================
// COMMON HEADER
// ======================================================
VO_Frame.Data[0] := VI_Slave_ID;
VO_Frame.Data[1] := L_Function_Byte;
VO_Frame.Data[2] := WORD_TO_BYTE(SHR(UINT_TO_WORD(VI_Start_Register), 8));
VO_Frame.Data[3] := WORD_TO_BYTE(UINT_TO_WORD(VI_Start_Register) AND 16#00FF);

CASE VI_Function_Code OF

    MB_FC03_READ_HOLDING_REGISTERS,
    MB_FC04_READ_INPUT_REGISTERS:

        VO_Frame.Data[4] := WORD_TO_BYTE(SHR(UINT_TO_WORD(VI_Register_Count), 8));
        VO_Frame.Data[5] := WORD_TO_BYTE(UINT_TO_WORD(VI_Register_Count) AND 16#00FF);

        VO_Frame.Length := 6;

    MB_FC06_WRITE_SINGLE_REGISTER:

        VO_Frame.Data[4] := WORD_TO_BYTE(SHR(VI_Write_Value[1], 8));
        VO_Frame.Data[5] := WORD_TO_BYTE(VI_Write_Value[1] AND 16#00FF);

        VO_Frame.Length := 6;

    MB_FC16_WRITE_MULTIPLE_REGISTERS:

        L_Byte_Count := VI_Register_Count * 2;

        IF L_Byte_Count > 64 THEN
            VO_Error := TRUE;
            VO_Error_Code := 16#0103;
            RETURN;
        END_IF;

        VO_Frame.Data[4] := WORD_TO_BYTE(SHR(UINT_TO_WORD(VI_Register_Count), 8));
        VO_Frame.Data[5] := WORD_TO_BYTE(UINT_TO_WORD(VI_Register_Count) AND 16#00FF);
        VO_Frame.Data[6] := UINT_TO_BYTE(L_Byte_Count);

        L_Pos := 7;

        FOR L_i := 1 TO UINT_TO_INT(VI_Register_Count) DO
            VO_Frame.Data[L_Pos] := WORD_TO_BYTE(SHR(VI_Write_Value[L_i], 8));
            VO_Frame.Data[L_Pos + 1] := WORD_TO_BYTE(VI_Write_Value[L_i] AND 16#00FF);
            L_Pos := L_Pos + 2;
        END_FOR;

        VO_Frame.Length := 7 + L_Byte_Count;

ELSE
    VO_Error := TRUE;
    VO_Error_Code := 16#0104;
    RETURN;
END_CASE;

// ======================================================
// CRC APPEND
// ======================================================
L_CRC := F_Modbus_RTU_CRC16(
    VI_Data := VO_Frame.Data,
    VI_Length := VO_Frame.Length
);

VO_Frame.CRC := L_CRC;
VO_Frame.Data[VO_Frame.Length] := WORD_TO_BYTE(L_CRC AND 16#00FF);
VO_Frame.Data[VO_Frame.Length + 1] := WORD_TO_BYTE(SHR(L_CRC, 8));
VO_Frame.Length := VO_Frame.Length + 2;
VO_Frame.Valid := TRUE;

END_FUNCTION_BLOCK

(* ---- FB_Mode_Manager.st ---- *)
FUNCTION_BLOCK FB_Mode_Manager

VAR_INPUT
    VI_Is_Night : BOOL;
    VI_System_Time_MS : UDINT;
END_VAR

VAR_OUTPUT
    VO_Mode : E_Behavior_Mode;
    VO_Mode_Code : UDINT;
END_VAR

// default
VO_Mode := BEHAVIOR_HOME;
VO_Mode_Code := 0;

// simple logic (observe-only)
IF VI_Is_Night THEN
    VO_Mode := BEHAVIOR_NIGHT;
    VO_Mode_Code := 100;
END_IF;

(* ---- FB_MQTT_Runtime_Adapter.st ---- *)
FUNCTION_BLOCK FB_MQTT_Runtime_Adapter
VAR_INPUT
    VI_Enable : BOOL;
    VI_System_Time_MS : UDINT;
END_VAR
VAR
    L_Frame : ST_Runtime_Bus_Frame;
    L_TX_Index : UINT;
END_VAR

IF NOT VI_Enable THEN
    RETURN;
END_IF;

L_TX_Index := UDINT_TO_UINT(GVL_Runtime_Bus.G_Last_Sequence_Id);

IF (L_TX_Index >= 1)
   AND (L_TX_Index <= 128) THEN

    L_Frame := GVL_Runtime_Bus.G_TX_Frames[L_TX_Index];

    IF L_Frame.Frame_Valid THEN

        IF GVL_Distributed_Authority.G_Distributed_Safety_Barrier_OK
           AND NOT GVL_Runtime_Sessions.G_Any_Stale_Session THEN

            L_Frame.Frame_Ack_Received := TRUE;
            L_Frame.Replication_Consistent := TRUE;
            L_Frame.Status_Code := 0;

        ELSE

            L_Frame.Replication_Rejected := TRUE;
            L_Frame.Status_Code := 2;

        END_IF;

        GVL_Runtime_Bus.G_TX_Frames[L_TX_Index] := L_Frame;

    END_IF;

END_IF;

END_FUNCTION_BLOCK

(* ---- FB_NVRAM_Manager.st ---- *)
FUNCTION_BLOCK FB_NVRAM_Manager
VAR_INPUT
    VI_Command                  : BYTE; // 1=WRITE, 2=READ
    VI_Offset                   : UDINT; // Смещение в байтах
    VI_DataRef                  : REFERENCE TO BYTE;
    VI_DataSize                 : UDINT; // КРИТИЧНО: используем этот размер вместо SIZEOF
    VI_System_Time_MS           : UDINT;
    VI_Operator_ID              : STRING(10);
    VI_IsActivePLC              : BOOL;
    VI_TwoPersonConfirmation    : BOOL;
END_VAR
VAR_OUTPUT
    VO_Done                     : BOOL;
    VO_Error                    : BOOL;
    VO_ErrorID                  : UDINT;
    // VO_ReadDataRef removed (REFERENCE TO not allowed in output)
    VO_HMI_Status_Message       : STRING(200);
END_VAR
VAR
    L_prev_Command              : BYTE;
    L_cmd_rising                : BOOL;
    L_i                         : UDINT;
    L_Data_Changed              : BOOL; // Флаг изменения данных
    L_pData                      : POINTER TO BYTE;
END_VAR
VAR CONSTANT
    C_MAX_NVRAM_SIZE            : UDINT := 12800;
END_VAR

// Детекция фронта команды
L_cmd_rising := (VI_Command <> 0) AND (L_prev_Command = 0);
L_prev_Command := VI_Command;

IF L_cmd_rising THEN
    VO_Done := FALSE;
    VO_Error := FALSE;
    VO_ErrorID := 0;
    VO_HMI_Status_Message := '';

    // Валидация смещения
    IF VI_Offset >= C_MAX_NVRAM_SIZE THEN
        VO_Error := TRUE;
        VO_ErrorID := 16#1501;
        VO_HMI_Status_Message := 'NVRAM: Неверное смещение';
        VO_Done := TRUE;
        RETURN;
    END_IF;

    // Валидация указателя
    IF NOT __ISVALIDREF(VI_DataRef) THEN
        VO_Error := TRUE;
        VO_ErrorID := 16#150A;
        VO_HMI_Status_Message := 'NVRAM: Недействительная ссылка на данные';
        VO_Done := TRUE;
        RETURN;
    END_IF;

    L_pData := ADR(VI_DataRef);

    IF (VI_Offset + VI_DataSize) > C_MAX_NVRAM_SIZE THEN
        VO_Error := TRUE;
        VO_ErrorID := 16#150B;
        VO_HMI_Status_Message := 'NVRAM: Размер данных превышает доступный объем';
        VO_Done := TRUE;
        RETURN;
    END_IF;

    IF VI_Command = 1 THEN // ЗАПИСЬ (WRITE)
        IF NOT VI_IsActivePLC THEN
            VO_Error := TRUE;
            VO_ErrorID := 16#1509;
            VO_HMI_Status_Message := 'NVRAM: Запись запрещена (STANDBY)';
        ELSE
            // Проверка на изменение данных перед записью
            L_Data_Changed := FALSE;
            FOR L_i := 0 TO VI_DataSize - 1 DO
                IF GVL_Retain.G_NVRAM_Data[VI_Offset + L_i] <> L_pData[L_i] THEN
                    L_Data_Changed := TRUE;
                    EXIT;
                END_IF;
            END_FOR;

            IF L_Data_Changed THEN
                // Безопасное копирование (WRITE)
                FOR L_i := 0 TO VI_DataSize - 1 DO
                    GVL_Retain.G_NVRAM_Data[VI_Offset + L_i] := L_pData[L_i];
                END_FOR;
                VO_HMI_Status_Message := 'NVRAM: Данные успешно сохранены в RETAIN';
            ELSE
                VO_HMI_Status_Message := 'NVRAM: Данные не изменились, запись пропущена';
            END_IF;
        END_IF;
        VO_Done := TRUE;
    END_IF;
END_IF;

IF VI_Command = 0 THEN
    VO_Done := FALSE;
END_IF;
// >>> BULK_SYNC_ANCHOR: FB_NVRAM_Manager <<<

(* ---- FB_OPCUA_Runtime_Adapter.st ---- *)
FUNCTION_BLOCK FB_OPCUA_Runtime_Adapter
VAR_INPUT
    VI_Enable : BOOL;
    VI_System_Time_MS : UDINT;
END_VAR
VAR
    L_Frame : ST_Runtime_Bus_Frame;
    L_TX_Index : UINT;
END_VAR

IF NOT VI_Enable THEN
    RETURN;
END_IF;

L_TX_Index := UDINT_TO_UINT(GVL_Runtime_Bus.G_Last_Sequence_Id);

IF (L_TX_Index >= 1)
   AND (L_TX_Index <= 128) THEN

    L_Frame := GVL_Runtime_Bus.G_TX_Frames[L_TX_Index];

    IF L_Frame.Frame_Valid THEN

        IF GVL_Distributed_Authority.G_Distributed_Safety_Barrier_OK
           AND NOT GVL_Runtime_Discovery.G_Any_Node_Quarantined THEN

            L_Frame.Frame_Ack_Received := TRUE;
            L_Frame.Replication_Consistent := TRUE;
            L_Frame.Status_Code := 0;

        ELSE

            L_Frame.Replication_Rejected := TRUE;
            L_Frame.Status_Code := 2;

        END_IF;

        GVL_Runtime_Bus.G_TX_Frames[L_TX_Index] := L_Frame;

    END_IF;

END_IF;

END_FUNCTION_BLOCK

(* ---- FB_Outdoor_Lighting_Controller.st ---- *)
FUNCTION_BLOCK FB_Outdoor_Lighting_Controller
VAR_INPUT
    VI_Ambient_Lux : REAL;
    VI_Motion      : BOOL;
    VI_Security    : BOOL;
END_VAR
VAR_OUTPUT
    VO_Light_On    : BOOL;
END_VAR

IF VI_Security AND VI_Motion THEN
    VO_Light_On := TRUE; // Тревожное освещение
ELSIF VI_Ambient_Lux < 50.0 THEN
    VO_Light_On := TRUE; // Ночное освещение
ELSE
    VO_Light_On := FALSE;
END_IF;

(* ---- FB_Ownership_Watchdog.st ---- *)
FUNCTION_BLOCK FB_Ownership_Watchdog
VAR_INPUT
    VI_Gas_Level : REAL;
    VI_Gas_Alarm : BOOL;
    VI_Leak_Alarm : BOOL;
    VI_Smoke_Alarm : BOOL;
END_VAR
VAR_OUTPUT
    VO_Ownership_Violation : BOOL;
END_VAR
VAR
    L_Last_Gas_Alarm : BOOL;
    L_Last_Leak_Alarm : BOOL;
    L_Last_Smoke_Alarm : BOOL;
END_VAR

VO_Ownership_Violation := FALSE;

// Gas: signal present, alarm disappeared
IF (VI_Gas_Level > 20.0) AND L_Last_Gas_Alarm AND (NOT VI_Gas_Alarm) THEN
    VO_Ownership_Violation := TRUE;
END_IF;

// Leak: once latched should not drop instantly
IF L_Last_Leak_Alarm AND (NOT VI_Leak_Alarm) THEN
    VO_Ownership_Violation := TRUE;
END_IF;

// Smoke: same rule
IF L_Last_Smoke_Alarm AND (NOT VI_Smoke_Alarm) THEN
    VO_Ownership_Violation := TRUE;
END_IF;

L_Last_Gas_Alarm := VI_Gas_Alarm;
L_Last_Leak_Alarm := VI_Leak_Alarm;
L_Last_Smoke_Alarm := VI_Smoke_Alarm;
END_FUNCTION_BLOCK

(* ---- FB_Periodic_Due_Gate.st ---- *)
FUNCTION_BLOCK FB_Periodic_Due_Gate
VAR_INPUT
    VI_Enable : BOOL;
    VI_Now_MS : UDINT;
    VI_Interval_MS : UDINT;
END_VAR
VAR_OUTPUT
    VO_Due : BOOL;
    VO_Last_Run_MS : UDINT;
END_VAR
VAR
    L_Elapsed_MS : UDINT;
    L_Interval_MS : UDINT;
END_VAR

VO_Due := FALSE;

IF NOT VI_Enable THEN
    RETURN;
END_IF;

L_Interval_MS := VI_Interval_MS;
IF L_Interval_MS = 0 THEN
    L_Interval_MS := 1;
END_IF;

IF VO_Last_Run_MS = 0 THEN
    VO_Last_Run_MS := VI_Now_MS;
    VO_Due := TRUE;
    RETURN;
END_IF;

IF VI_Now_MS >= VO_Last_Run_MS THEN
    L_Elapsed_MS := VI_Now_MS - VO_Last_Run_MS;
ELSE
    L_Elapsed_MS := (4294967295 - VO_Last_Run_MS) + VI_Now_MS + 1;
END_IF;

IF L_Elapsed_MS >= L_Interval_MS THEN
    VO_Due := TRUE;
    VO_Last_Run_MS := VI_Now_MS;
END_IF;

END_FUNCTION_BLOCK
// >>> BULK_SYNC_ANCHOR: FB_Periodic_Due_Gate <<<

(* ---- FB_Persist_Builder.st ---- *)
FUNCTION_BLOCK FB_Persist_Builder
VAR_INPUT
    VI_State : ST_System_State;
END_VAR

VAR_IN_OUT
    VIO_PersistStruct : ST_Persist;
END_VAR

// === BUILD STRUCT FROM STATE ===
// === NVRAM SNAPSHOT VIA STRUCT ADAPTER ===
L_Persist_Struct.System_Mode := GVL_STATE.G_System_Mode;

L_Persist_Struct.Safety_Gas_Latched := GVL_STATE.G_Safety_Gas_Latched;
L_Persist_Struct.Safety_Smoke_Latched := GVL_STATE.G_Safety_Smoke_Latched;
L_Persist_Struct.Safety_Leak_Latched := GVL_STATE.G_Safety_Leak_Latched;

L_Persist_Struct.DHW_Heating_Pump := GVL_STATE.G_DHW_Heating_Pump;
L_Persist_Struct.Valid := TRUE;

// mirror to legacy persistent variables
GVL_PERSISTENT.P_System_Mode := L_Persist_Struct.System_Mode;

GVL_PERSISTENT.P_Safety_Gas_Latched := L_Persist_Struct.Safety_Gas_Latched;
GVL_PERSISTENT.P_Safety_Smoke_Latched := L_Persist_Struct.Safety_Smoke_Latched;
GVL_PERSISTENT.P_Safety_Leak_Latched := L_Persist_Struct.Safety_Leak_Latched;

GVL_PERSISTENT.P_DHW_Heating_Active := L_Persist_Struct.DHW_Heating_Pump;
GVL_PERSISTENT.P_Valid := L_Persist_Struct.Valid;

(* ---- FB_Persist_Pipeline.st ---- *)
FUNCTION_BLOCK FB_Persist_Pipeline
VAR_INPUT
    VI_PersistStruct : ST_Persist;
    VI_System_Time_MS : UDINT;
    VI_IsActivePLC : BOOL;
END_VAR
VAR_IN_OUT
    VIO_Apply_Settings : BOOL;
    VIO_Persist_Buffer : ARRAY[0..4] OF BYTE;
    VIO_Last_Written_Persist_Buffer : ARRAY[0..4] OF BYTE;
    VIO_Last_Persist_Write_MS : UDINT;
END_VAR
VAR_OUTPUT
    VO_NVRAM_Cmd : BYTE;
    VO_NVRAM_Offset : UDINT;
    VO_NVRAM_Done : BOOL;
    VO_NVRAM_Err : BOOL;
    VO_NVRAM_ErrID : UDINT;
END_VAR
VAR
    fbNVRAMManager : FB_NVRAM_Manager;
    L_Persist_Buffer_Changed : BOOL;
END_VAR

// === SERIALIZE PERSIST STRUCT → BUFFER ===

// System Mode
VIO_Persist_Buffer[0] := TO_BYTE(TO_INT(VI_PersistStruct.System_Mode));

// Gas
IF VI_PersistStruct.Safety_Gas_Latched THEN
    VIO_Persist_Buffer[1] := BYTE#1;
ELSE
    VIO_Persist_Buffer[1] := BYTE#0;
END_IF;

// Smoke
IF VI_PersistStruct.Safety_Smoke_Latched THEN
    VIO_Persist_Buffer[2] := BYTE#1;
ELSE
    VIO_Persist_Buffer[2] := BYTE#0;
END_IF;

// Leak
IF VI_PersistStruct.Safety_Leak_Latched THEN
    VIO_Persist_Buffer[3] := BYTE#1;
ELSE
    VIO_Persist_Buffer[3] := BYTE#0;
END_IF;

// DHW Pump
IF VI_PersistStruct.DHW_Heating_Pump THEN
    VIO_Persist_Buffer[4] := BYTE#1;
ELSE
    VIO_Persist_Buffer[4] := BYTE#0;
END_IF;

// === END SERIALIZE ===

L_Persist_Buffer_Changed :=
    (VIO_Persist_Buffer[0] <> VIO_Last_Written_Persist_Buffer[0]) OR
    (VIO_Persist_Buffer[1] <> VIO_Last_Written_Persist_Buffer[1]) OR
    (VIO_Persist_Buffer[2] <> VIO_Last_Written_Persist_Buffer[2]) OR
    (VIO_Persist_Buffer[3] <> VIO_Last_Written_Persist_Buffer[3]) OR
    (VIO_Persist_Buffer[4] <> VIO_Last_Written_Persist_Buffer[4]);

VO_NVRAM_Cmd := 0;
VO_NVRAM_Offset := 0;

IF VIO_Apply_Settings THEN
    // explicit config apply may request a controlled write
    VO_NVRAM_Cmd := 1;
    VIO_Apply_Settings := FALSE;

ELSIF L_Persist_Buffer_Changed THEN
    // controlled write: no more often than once per 60 seconds
    IF (VIO_Last_Persist_Write_MS = 0) OR
       ((VI_System_Time_MS - VIO_Last_Persist_Write_MS) >= 60000) THEN
        VO_NVRAM_Cmd := 1;
    END_IF;
END_IF;

fbNVRAMManager(
    VI_Command := VO_NVRAM_Cmd,
    VI_Offset := VO_NVRAM_Offset,
    VI_DataRef := VIO_Persist_Buffer[0],
    VI_DataSize := 5,
    VI_System_Time_MS := VI_System_Time_MS,
    VI_Operator_ID := 'SYSTEM',
    VI_IsActivePLC := VI_IsActivePLC,
    VI_TwoPersonConfirmation := FALSE,
    VO_Done => VO_NVRAM_Done,
    VO_Error => VO_NVRAM_Err,
    VO_ErrorID => VO_NVRAM_ErrID
);

IF (VO_NVRAM_Cmd = 1) AND VO_NVRAM_Done AND NOT VO_NVRAM_Err THEN
    VIO_Last_Written_Persist_Buffer[0] := VIO_Persist_Buffer[0];
    VIO_Last_Written_Persist_Buffer[1] := VIO_Persist_Buffer[1];
    VIO_Last_Written_Persist_Buffer[2] := VIO_Persist_Buffer[2];
    VIO_Last_Written_Persist_Buffer[3] := VIO_Persist_Buffer[3];
    VIO_Last_Written_Persist_Buffer[4] := VIO_Persist_Buffer[4];
    VIO_Last_Persist_Write_MS := VI_System_Time_MS;
END_IF;

(* ---- FB_PID_Controller.st ---- *)
FUNCTION_BLOCK FB_PID_Controller
VAR_INPUT
    VI_SetPoint : REAL;
    VI_ProcessValue : REAL;
    VI_Kp : REAL;
    VI_Tn : REAL;
    VI_Tv : REAL;
    VI_Y_Min : REAL := 0.0;
    VI_Y_Max : REAL := 100.0;
    VI_Manual_Mode : BOOL;
    VI_Manual_Value : REAL;
    VI_Deadband : REAL := 0.1;
    VI_Cycle_Time_S : REAL := 0.01;
    VI_Reset : BOOL;
END_VAR
VAR_OUTPUT
    VO_Output : REAL;
    VO_Error : REAL;
    VO_Limiting : BOOL;
END_VAR
VAR
    L_Integral_Sum : REAL;
    L_Prev_Error : REAL;
    L_Derivative : REAL;
    L_P_Term : REAL;
    L_I_Candidate : REAL;
    L_D_Term : REAL;
    L_Output_Predicted : REAL;
    L_Output_Raw : REAL;
    L_Cycle_Time_Safe : REAL;
END_VAR

(* explicit cast for safety *)
L_Cycle_Time_Safe := REAL(VI_Cycle_Time_S);

END_FUNCTION_BLOCK

(* ---- FB_Predictive_Diagnostics_Runtime.st ---- *)
FUNCTION_BLOCK FB_Predictive_Diagnostics_Runtime
VAR_INPUT
    VI_Enable : BOOL;
    VI_System_Time_MS : UDINT;
END_VAR
VAR
    L_i : INT;
    L_State : ST_Predictive_Diagnostics_State;
    L_Feedback : ST_Water_Valve_Feedback_State;
    L_Recovery : ST_Water_Recovery_Runtime_State;

    L_Any_Degrading : BOOL;
    L_Any_Service : BOOL;
    L_Any_Urgent : BOOL;
END_VAR

IF NOT VI_Enable THEN
    GVL_Predictive_Diagnostics.G_Runtime_Valid := FALSE;
    RETURN;
END_IF;

FOR L_i := 1 TO GVL_CONSTANTS.C_MAX_FLOOD_SENSORS DO

    L_State := GVL_Predictive_Diagnostics.G_Diagnostics_State[L_i];

    L_Feedback :=
        GVL_Water_Valve_Feedback.G_Valve_Feedback_State[L_i];

    L_Recovery :=
        GVL_Water_Recovery_Runtime.G_Recovery_State[L_i];

    L_State.Runtime_Valid := TRUE;
    L_State.Runtime_System_Time_MS := VI_System_Time_MS;

    L_State.Device_Id := TO_UINT(L_i);
    L_State.Valve_Group_Id := L_Feedback.Valve_Group_Id;

    IF L_Feedback.Feedback_Timeout THEN
        L_State.Timeout_Count := L_State.Timeout_Count + 1;
    END_IF;

    IF L_Feedback.Feedback_Conflict THEN
        L_State.Conflict_Count := L_State.Conflict_Count + 1;
    END_IF;

    IF L_Recovery.Recovery_Denied THEN
        L_State.Recovery_Denied_Count :=
            L_State.Recovery_Denied_Count + 1;
    END_IF;

    L_State.Failure_Count :=
        L_State.Timeout_Count
        + L_State.Conflict_Count
        + L_State.Recovery_Denied_Count;

    // Predictive accumulation model foundation.
    L_State.Wear_Score :=
        TO_REAL(L_State.Failure_Count) * 0.1;

    L_State.Reliability_Score :=
        100.0 - L_State.Wear_Score;

    IF L_State.Reliability_Score < 0.0 THEN
        L_State.Reliability_Score := 0.0;
    END_IF;

    IF L_State.Failure_Count >= 3 THEN

        L_State.Degradation_Accumulating := TRUE;
        L_State.Service_Recommended := TRUE;

    END_IF;

    IF L_State.Failure_Count >= 10 THEN

        L_State.Service_Urgent := TRUE;
        L_State.Predictive_Quarantine_Recommended := TRUE;

    END_IF;

    IF L_State.Conflict_Count >= 2 THEN
        L_State.Intermittent_Fault_Suspected := TRUE;
    END_IF;

    IF L_State.Service_Urgent THEN

        L_State.Status_Code := 2;
        L_State.Status_Text :=
            'Urgent predictive maintenance required';

    ELSIF L_State.Service_Recommended THEN

        L_State.Status_Code := 1;
        L_State.Status_Text :=
            'Predictive maintenance recommended';

    ELSE

        L_State.Status_Code := 0;
        L_State.Status_Text :=
            'Predictive diagnostics healthy';

    END_IF;

    GVL_Predictive_Diagnostics.G_Diagnostics_State[L_i] :=
        L_State;

    L_Any_Degrading :=
        L_Any_Degrading
        OR L_State.Degradation_Accumulating;

    L_Any_Service :=
        L_Any_Service
        OR L_State.Service_Recommended;

    L_Any_Urgent :=
        L_Any_Urgent
        OR L_State.Service_Urgent;

END_FOR;

GVL_Predictive_Diagnostics.G_Any_Degradation_Accumulating :=
    L_Any_Degrading;

GVL_Predictive_Diagnostics.G_Any_Service_Recommended :=
    L_Any_Service;

GVL_Predictive_Diagnostics.G_Any_Urgent_Service :=
    L_Any_Urgent;

GVL_Predictive_Diagnostics.G_Runtime_Valid := TRUE;
GVL_Predictive_Diagnostics.G_Last_Update_MS := VI_System_Time_MS;

IF L_Any_Urgent THEN
    GVL_Predictive_Diagnostics.G_Status_Code := 2;
    GVL_Predictive_Diagnostics.G_Status_Text :=
        'Urgent predictive maintenance required';
ELSIF L_Any_Service THEN
    GVL_Predictive_Diagnostics.G_Status_Code := 1;
    GVL_Predictive_Diagnostics.G_Status_Text :=
        'Predictive maintenance recommended';
ELSE
    GVL_Predictive_Diagnostics.G_Status_Code := 0;
    GVL_Predictive_Diagnostics.G_Status_Text :=
        'Predictive diagnostics runtime healthy';
END_IF;

END_FUNCTION_BLOCK

(* ---- FB_Presence_Manager.st ---- *)
FUNCTION_BLOCK FB_Presence_Manager

VAR_INPUT
    VI_Motion_Sensors : ARRAY[1..32] OF BOOL;
    VI_System_Time_MS : UDINT;
END_VAR

VAR_OUTPUT
    VO_Any_Motion : BOOL;
    VO_Occupied : BOOL;
    VO_Auto_Away : BOOL;
    VO_Last_Motion_TS : UDINT;
END_VAR

VAR
    L_Last_Motion_TS : UDINT := 0;
    L_Initialized : BOOL := FALSE;
    L_Timeout_MS : UDINT := 900000; // 15 min away delay
    L_i : INT;
END_VAR

// detect any motion
VO_Any_Motion := FALSE;
FOR L_i := 1 TO 32 DO
    IF VI_Motion_Sensors[L_i] THEN
        VO_Any_Motion := TRUE;
    END_IF;
END_FOR;

// init protection (avoid instant AWAY at boot)
IF NOT L_Initialized THEN
    L_Last_Motion_TS := VI_System_Time_MS;
    L_Initialized := TRUE;
END_IF;

// fast return: any motion immediately updates timestamp
IF VO_Any_Motion THEN
    L_Last_Motion_TS := VI_System_Time_MS;
END_IF;

// hysteresis logic:
// stay OCCUPIED until timeout expires
IF (VI_System_Time_MS - L_Last_Motion_TS) < L_Timeout_MS THEN
    VO_Occupied := TRUE;
ELSE
    VO_Occupied := FALSE;
END_IF;

VO_Auto_Away := NOT VO_Occupied;
VO_Last_Motion_TS := L_Last_Motion_TS;
END_FUNCTION_BLOCK

(* ---- FB_Presence_Playback.st ---- *)
FUNCTION_BLOCK FB_Presence_Playback
VAR_INPUT
    VI_Mode_Record : BOOL;
    VI_Time_Index   : UDINT;
END_VAR
VAR_IN_OUT
    VI_Light_Inputs : ARRAY[1..32] OF BOOL;
END_VAR
VAR_OUTPUT
    VO_Light_Outputs : ARRAY[1..32] OF BOOL;
END_VAR
VAR
    L_Current_Slot : UDINT;
    L_i : INT;
END_VAR

L_Current_Slot := (VI_Time_Index / (GVL_CONSTANTS.C_MS_IN_MINUTE * 10)) MOD TO_UDINT(GVL_CONSTANTS.C_MAX_PRESENCE_HISTORY);

FOR L_i := 1 TO 32 DO
    VO_Light_Outputs[L_i] := FALSE;
END_FOR;

IF VI_Mode_Record THEN
    GVL_Retain.G_Presence_History[L_Current_Slot] := 0;
    FOR L_i := 1 TO 16 DO
        IF VI_Light_Inputs[L_i] THEN
            GVL_Retain.G_Presence_History[L_Current_Slot] :=
                GVL_Retain.G_Presence_History[L_Current_Slot] OR SHL(WORD#1, L_i - 1);
        END_IF;
    END_FOR;
ELSE
    FOR L_i := 1 TO 16 DO
        VO_Light_Outputs[L_i] :=
            (GVL_Retain.G_Presence_History[L_Current_Slot] AND SHL(WORD#1, L_i - 1)) <> 0;
    END_FOR;
END_IF;

END_FUNCTION_BLOCK

(* ---- FB_Random_Generator.st ---- *)
FUNCTION_BLOCK FB_Random_Generator
VAR
    L_seed : UDINT := 1;
    L_Is_Seeded : BOOL := FALSE;
END_VAR
VAR CONSTANT
    C_LCG_MULTIPLIER : UDINT := 1664525;
    C_LCG_INCREMENT  : UDINT := 1013904223;
    C_LCG_MODULUS    : LREAL := 4294967296.0;
END_VAR

METHOD Seed : BOOL
VAR_INPUT
    VI_Seed_Value : UDINT;
END_VAR
L_seed := VI_Seed_Value;
L_Is_Seeded := TRUE;
Seed := TRUE;
END_METHOD

METHOD Random_Int_Range : UDINT
VAR_INPUT
    VI_min : UDINT;
    VI_max : UDINT;
    VI_System_Time_MS : UDINT; // Для автоматического сидирования
END_VAR
VAR
    L_range : UDINT;
    L_rand_factor : LREAL;
END_VAR

IF NOT L_Is_Seeded AND VI_System_Time_MS > 0 THEN
    L_seed := VI_System_Time_MS;
    L_Is_Seeded := TRUE;
END_IF;

L_seed := (C_LCG_MULTIPLIER * L_seed) + C_LCG_INCREMENT;

IF VI_max > VI_min THEN
        L_range := VI_max - VI_min;
        // Используем LREAL для точности и исключения выхода за границу
        L_rand_factor := TO_LREAL(L_seed) / C_LCG_MODULUS;
        Random_Int_Range := VI_min + TO_UDINT(L_rand_factor * TO_LREAL(L_range + 1));

        // Финальная защита от переполнения
        IF Random_Int_Range > VI_max THEN
            Random_Int_Range := VI_max;
        END_IF;
    ELSE
        Random_Int_Range := VI_min;
    END_IF;
